    TEXT549 : BOOL ;	//TEXT N.549
    TEXT550 : BOOL ;	//TEXT N.550
    TEXT551 : BOOL ;	//TEXT N.551
    TEXT552 : BOOL ;	//TEXT N.552
    TEXT569 : BOOL ;	//TEXT N.569
    TEXT570 : BOOL ;	//TEXT N.570
    TEXT571 : BOOL ;	//TEXT N.571
    TEXT572 : BOOL ;	//TEXT N.572
    TEXT573 : BOOL ;	//TEXT N.573
    TEXT574 : BOOL ;	//TEXT N.574
    TEXT575 : BOOL ;	//TEXT N.575
    TEXT576 : BOOL ;	//TEXT N.576
    TEXT561 : BOOL ;	//TEXT N.561
    TEXT562 : BOOL ;	//TEXT N.562
    TEXT563 : BOOL ;	//TEXT N.563
    TEXT564 : BOOL ;	//TEXT N.564
    TEXT565 : BOOL ;	//TEXT N.565
    TEXT566 : BOOL ;	//TEXT N.566
    TEXT567 : BOOL ;	//TEXT N.567
    TEXT568 : BOOL ;	//TEXT N.568
    TEXT585 : BOOL ;	//TEXT N.585
    TEXT586 : BOOL ;	//TEXT N.586
    TEXT587 : BOOL ;	//TEXT N.587
    TEXT588 : BOOL ;	//TEXT N.588
    TEXT589 : BOOL ;	//TEXT N.589
    TEXT590 : BOOL ;	//TEXT N.590
    TEXT591 : BOOL ;	//TEXT N.591
    TEXT592 : BOOL ;	//TEXT N.592
    TEXT577 : BOOL ;	//TEXT N.577
    TEXT578 : BOOL ;	//TEXT N.578
    TEXT579 : BOOL ;	//TEXT N.579
    TEXT580 : BOOL ;	//TEXT N.580
    TEXT581 : BOOL ;	//TEXT N.581
    TEXT582 : BOOL ;	//TEXT N.582
    TEXT583 : BOOL ;	//TEXT N.583
    TEXT584 : BOOL ;	//TEXT N.584
    TEXT601 : BOOL ;	//TEXT N.601
    TEXT602 : BOOL ;	//TEXT N.602
    TEXT603 : BOOL ;	//TEXT N.603
    TEXT604 : BOOL ;	//TEXT N.604
    TEXT605 : BOOL ;	//TEXT N.605
    TEXT606 : BOOL ;	//TEXT N.606
    TEXT607 : BOOL ;	//TEXT N.607
    TEXT608 : BOOL ;	//TEXT N.608
    TEXT593 : BOOL ;	//TEXT N.593
    TEXT594 : BOOL ;	//TEXT N.594
    TEXT595 : BOOL ;	//TEXT N.595
    TEXT596 : BOOL ;	//TEXT N.596
    TEXT597 : BOOL ;	//TEXT N.597
    TEXT598 : BOOL ;	//TEXT N.598
    TEXT599 : BOOL ;	//TEXT N.599
    TEXT600 : BOOL ;	//TEXT N.600
    TEXT617 : BOOL ;	//TEXT N.617
    TEXT618 : BOOL ;	//TEXT N.618
    TEXT619 : BOOL ;	//TEXT N.619
    TEXT620 : BOOL ;	//TEXT N.620
    TEXT621 : BOOL ;	//TEXT N.621
    TEXT622 : BOOL ;	//TEXT N.622
    TEXT623 : BOOL ;	//TEXT N.623
    TEXT624 : BOOL ;	//TEXT N.624
    TEXT609 : BOOL ;	//TEXT N.609
    TEXT610 : BOOL ;	//TEXT N.610
    TEXT611 : BOOL ;	//TEXT N.611
    TEXT612 : BOOL ;	//TEXT N.612
    TEXT613 : BOOL ;	//TEXT N.613
    TEXT614 : BOOL ;	//TEXT N.614
    TEXT615 : BOOL ;	//TEXT N.615
    TEXT616 : BOOL ;	//TEXT N.616
    TEXT633 : BOOL ;	//TEXT N.633
    TEXT634 : BOOL ;	//TEXT N.634
    TEXT635 : BOOL ;	//TEXT N.635
    TEXT636 : BOOL ;	//TEXT N.636
    TEXT637 : BOOL ;	//TEXT N.637
    TEXT638 : BOOL ;	//TEXT N.638
    TEXT639 : BOOL ;	//TEXT N.639
    TEXT640 : BOOL ;	//TEXT N.640
    TEXT625 : BOOL ;	//TEXT N.625
    TEXT626 : BOOL ;	//TEXT N.626
    TEXT627 : BOOL ;	//TEXT N.627
    TEXT628 : BOOL ;	//TEXT N.628
    TEXT629 : BOOL ;	//TEXT N.629
    TEXT630 : BOOL ;	//TEXT N.630
    TEXT631 : BOOL ;	//TEXT N.631
    TEXT632 : BOOL ;	//TEXT N.632
   END_STRUCT ;
   PaginaDaVisualizzare : INT ;	//Number of page to display
   PaginaPrecedenteSetup : INT ;	//Number of page displayed before "Setup" page
   NumeroComandoManuale : INT ;	//Number of manual command
   BoschProgramManuale : BYTE ;	//Number of program of screwdriver in manual mode
   ServiceAsseSelezionato : BYTE ;	//Axis selected for movement in service mode (0=X; 1=Y; 2=Z; 3=C; 4=P)
   ServiceTipoJog : BYTE ;	//Kind of jog movement in service mode (0=continue; 1=incremental)
   ServiceFieldsDisplayed : BYTE ;	//Identify the fields to be displayed in service page
   TypePointTeachIn : BYTE ;	//Kind of screw in teach-in mode
   PointWeldingTeachIn : BYTE ;	//Identification of the screw in tech-in mode
   TeachInFieldsDisplayed : STRUCT 	//Identify the fields to be displayed in teach-in page
    Punto1Saldatura : BOOL ;
    Punto2Saldatura : BOOL ;
    Punto3Saldatura : BOOL ;
    Punto4Saldatura : BOOL ;
    Punto5Saldatura : BOOL ;
    Punto6Saldatura : BOOL ;
    Punto7Saldatura : BOOL ;
    Punto8Saldatura : BOOL ;
    Punto9Saldatura : BOOL ;
    Punto10Saldatura : BOOL ;
    Punto11Saldatura : BOOL ;
    Punto12Saldatura : BOOL ;
    Punto13Saldatura : BOOL ;
    PuntoVisione : BOOL ;
    Riserva1 : BOOL ;
    Riserva2 : BOOL ;
   END_STRUCT ;
   Target_Inc : DINT ;	//Target for the incremental movement
  END_STRUCT ;	
BEGIN
END_DATA_BLOCK

DATA_BLOCK "Timer"	// DB 20
VERSION : 0.1
  STRUCT
   TmrOutGas : S5TIME  := S5T#1M;
   TmrIgnition : S5TIME  := S5T#20S;
   TmrDelayWelding : S5TIME  := S5T#300MS;
   time1 : S5TIME ;
   time11 : S5TIME ;
   time12 : S5TIME ;
   time13 : S5TIME ;
   time14 : S5TIME ;
   time15 : S5TIME ;
   time16 : S5TIME ;
   time17 : S5TIME ;
   time18 : S5TIME ;
   time19 : S5TIME ;
   time110 : S5TIME ;
   time111 : S5TIME ;
   time112 : S5TIME ;
   time113 : S5TIME ;
   time114 : S5TIME ;
   time115 : S5TIME ;
   time116 : S5TIME ;
   Override : INT  := 20;
   riserva : INT ;
   riserva2 : INT ;
   Comp01_OK : BOOL ;
   Comp02_OK : BOOL ;
   Comp03_OK : BOOL ;
   Comp04_OK : BOOL ;
   Comp05_OK : BOOL ;
   Comp06_OK : BOOL ;
   Comp07_OK : BOOL ;
   Comp08_OK : BOOL ;
   Comp09_OK : BOOL ;
   Comp10_OK : BOOL ;
   Comp11_OK : BOOL ;
   Comp12_OK : BOOL ;
   Comp13_OK : BOOL ;
   Comp14_OK : BOOL ;
   Comp15_OK : BOOL ;
   Comp16_OK : BOOL ;
   OffsetX1 : DINT ;
   OffsetY1 : DINT ;
   okAletta1 : BOOL ;
   okAletta2 : BOOL ;
   okAletta3 : BOOL ;
   okAletta4 : BOOL ;
   okAletta5 : BOOL ;
   okAletta6 : BOOL ;
   okAletta7 : BOOL ;
   okAletta8 : BOOL ;
   okAletta9 : BOOL ;
   okAletta10 : BOOL ;
   okAletta11 : BOOL ;
   okAletta12 : BOOL ;
   okAletta13 : BOOL ;
   okAletta14 : BOOL ;
   okAletta15 : BOOL ;
   okAletta16 : BOOL ;
   okAletta17 : BOOL ;
   okAletta18 : BOOL ;
   okAletta19 : BOOL ;
   okAletta20 : BOOL ;
   CheckComponent : BOOL  := TRUE;	//Check component with tool 1 --> Disable ; 0 --> Enable
   CheckTelec : BOOL ;	//Check Component with Omron 1 --> Disable ; 0 --> Enable
   check1 : BOOL ;
   CheckTelecafter : BOOL ;	//Check Component with Omron 1 --> Disable ; 0 --> Enable
   okAletta1_PP : BOOL ;
   okAletta2_PP : BOOL ;
   okAletta3_PP : BOOL ;
   okAletta4_PP : BOOL ;
   okAletta5_PP : BOOL ;
   okAletta6_PP : BOOL ;
   okAletta7_PP : BOOL ;
   okAletta8_PP : BOOL ;
   okAletta9_PP : BOOL ;
   okAletta10_PP : BOOL ;
   okAletta11_PP : BOOL ;
   okAletta12_PP : BOOL ;
   okAletta13_PP : BOOL ;
   okAletta14_PP : BOOL ;
   okAletta15_PP : BOOL ;
   okAletta16_PP : BOOL ;
   okAletta17_PP : BOOL ;
   okAletta18_PP : BOOL ;
   okAletta19_PP : BOOL ;
   okAletta20_PP : BOOL ;
   NumberVane : INT ;
  END_STRUCT ;	
BEGIN
   TmrOutGas := S5T#1M;
   TmrIgnition := S5T#20S;
   TmrDelayWelding := S5T#300MS;
   Override := 100;
   OffsetX1 := L#350;
   OffsetY1 := L#400;
END_DATA_BLOCK

DATA_BLOCK "DBWork"	// DB 21
TITLE = Recipe of part in production
VERSION : 0.1
  STRUCT
   Famiglia : BYTE  := B#16#2;	//Type of family of product(2=Step2; 3=Step3)
   Turbo : BYTE  := B#16#1;	//Type of product
   Portapezzo1 : INT  := 1;	//Code of work rest 1
   Portapezzo2 : INT  := 1;	//Code of work rest 2
   TempoSaldatura : ARRAY  [1 .. 20 ] OF STRUCT
    Tempo : S5TIME  := S5T#1S;
   END_STRUCT ;
   CoordSaldatura : ARRAY  [1 .. 20 ] OF //Coordinates of points
   STRUCT
    X1 : DINT ;	//X coordinate of point
    Y1 : DINT ;	//Y coordinate of point
    X2 : DINT ;
    Y2 : DINT ;
   END_STRUCT ;
   EnableTelecamera : BOOL  := TRUE;
   PP : ARRAY  [1 .. 2 ] OF STRUCT
    Vuoto : BOOL ;
    Caricato : BOOL ;
    Bloccato : BOOL ;
    Fuori : BOOL ;
    Dentro : BOOL ;
    InLavorazione : BOOL ;
    Lavorato : BOOL ;
    Buono : BOOL ;
    Scarto : BOOL ;
    NumSaldaturaAtt : INT ;
   END_STRUCT ;
   NumeroAnomalie : DINT ;
   NumeroPezziProd : DINT ;
   NumeroSaldature : INT ;
   Riserva : DINT ;	//position X for camera check
   Riserva1 : DINT ;	//position Y for camera check
   RotationTable : BOOL ;	//angle rotation 1-->PP1 on welding; 0-->PP2 on Welding
   PointCamCheck : ARRAY  [1 .. 10 ] OF STRUCT
    x : DINT ;
    y : DINT ;
   END_STRUCT ;
  END_STRUCT ;	
BEGIN
   Famiglia := B#16#2;
   Turbo := B#16#1;
   Portapezzo1 := 1;
   Portapezzo2 := 1;
   TempoSaldatura[1].Tempo := S5T#1S;
   TempoSaldatura[2].Tempo := S5T#2S;
   TempoSaldatura[3].Tempo := S5T#1S;
   TempoSaldatura[4].Tempo := S5T#1S;
   TempoSaldatura[5].Tempo := S5T#1S;
   TempoSaldatura[6].Tempo := S5T#1S;
   TempoSaldatura[7].Tempo := S5T#1S;
   TempoSaldatura[8].Tempo := S5T#1S;
   TempoSaldatura[9].Tempo := S5T#1S;
   TempoSaldatura[10].Tempo := S5T#1S;
   TempoSaldatura[11].Tempo := S5T#1S;
   TempoSaldatura[12].Tempo := S5T#1S;
   TempoSaldatura[13].Tempo := S5T#1S;
   TempoSaldatura[14].Tempo := S5T#1S;
   TempoSaldatura[15].Tempo := S5T#1S;
   TempoSaldatura[16].Tempo := S5T#1S;
   TempoSaldatura[17].Tempo := S5T#1S;
   TempoSaldatura[18].Tempo := S5T#1S;
   TempoSaldatura[19].Tempo := S5T#1S;
   TempoSaldatura[20].Tempo := S5T#1S;
   CoordSaldatura[1].X1 := L#-60766;
   CoordSaldatura[1].Y1 := L#-86096;
   CoordSaldatura[1].X2 := L#-60406;
   CoordSaldatura[1].Y2 := L#-86246;
   CoordSaldatura[2].X1 := L#-46600;
   CoordSaldatura[2].Y1 := L#-81431;
   CoordSaldatura[2].X2 := L#-46422;
   CoordSaldatura[2].Y2 := L#-81523;
   CoordSaldatura[3].X1 := L#-29709;
   CoordSaldatura[3].Y1 := L#-81739;
   CoordSaldatura[3].X2 := L#-29405;
   CoordSaldatura[3].Y2 := L#-81809;
   CoordSaldatura[4].X1 := L#-16402;
   CoordSaldatura[4].Y1 := L#-86931;
   CoordSaldatura[4].X2 := L#-116220;
   CoordSaldatura[4].Y2 := L#-86961;
   CoordSaldatura[5].X1 := L#-11762;
   CoordSaldatura[5].Y1 := L#-95066;
   CoordSaldatura[5].X2 := L#-11500;
   CoordSaldatura[5].Y2 := L#-95199;
   CoordSaldatura[6].X1 := L#-17500;
   CoordSaldatura[6].Y1 := L#-102971;
   CoordSaldatura[6].X2 := L#-17415;
   CoordSaldatura[6].Y2 := L#-103088;
   CoordSaldatura[7].X1 := L#-31505;
   CoordSaldatura[7].Y1 := L#-107714;
   CoordSaldatura[7].X2 := L#-31400;
   CoordSaldatura[7].Y2 := L#-108200;
   CoordSaldatura[8].X1 := L#-48449;
   CoordSaldatura[8].Y1 := L#-107375;
   CoordSaldatura[8].X2 := L#-48367;
   CoordSaldatura[8].Y2 := L#-107501;
   CoordSaldatura[9].X1 := L#-61760;
   CoordSaldatura[9].Y1 := L#-102188;
   CoordSaldatura[9].X2 := L#-61561;
   CoordSaldatura[9].Y2 := L#-102300;
   CoordSaldatura[10].X1 := L#-66400;
   CoordSaldatura[10].Y1 := L#-94028;
   CoordSaldatura[10].Y2 := L#-94249;
   EnableTelecamera := TRUE;
END_DATA_BLOCK

DATA_BLOCK "coordinate"	// DB 22
VERSION : 0.1
  STRUCT
   CoordSaldaturaPP1 : ARRAY  [1 .. 20 ] OF //Coordinates of points
   STRUCT
    X1 : DINT ;	//X coordinate of point PP1
    Y1 : DINT ;	//Y coordinate of point PP1
    X2 : DINT ;
    Y2 : DINT ;
   END_STRUCT ;
   CoordSaldaturaPP2 : ARRAY  [1 .. 20 ] OF //Coordinates of points
   STRUCT
    X1 : DINT ;	//X coordinate of point PP2
    Y1 : DINT ;	//Y coordinate of point PP2
    X2 : DINT ;
    Y2 : DINT ;
   END_STRUCT ;
   CoordSaldaturaPP3 : ARRAY  [1 .. 20 ] OF //Coordinates of points
   STRUCT
    X1 : DINT ;	//X coordinate of point PP3
    Y1 : DINT ;	//Y coordinate of point PP3
    X2 : DINT ;
    Y2 : DINT ;
   END_STRUCT ;
   CoordSaldaturaPP4 : ARRAY  [1 .. 20 ] OF //Coordinates of points
   STRUCT
    X1 : DINT ;	//X coordinate of point PP4
    Y1 : DINT ;	//Y coordinate of point PP4
    X2 : DINT ;
    Y2 : DINT ;
   END_STRUCT ;
   CoordSaldaturaPP5 : ARRAY  [1 .. 20 ] OF //Coordinates of points
   STRUCT
    X1 : DINT ;	//X coordinate of point PP5
    Y1 : DINT ;	//Y coordinate of point PP5
    X2 : DINT ;
    Y2 : DINT ;
   END_STRUCT ;
   CoordSaldaturaPP6 : ARRAY  [1 .. 20 ] OF STRUCT
    X1 : DINT ;
    Y1 : DINT ;
    X2 : DINT ;
    Y2 : DINT ;
   END_STRUCT ;
   CoordSaldaturaPP7 : ARRAY  [1 .. 20 ] OF STRUCT
    X1 : DINT ;
    Y1 : DINT ;
    X2 : DINT ;
    Y2 : DINT ;
   END_STRUCT ;
   CoordSaldaturaPP8 : ARRAY  [1 .. 20 ] OF STRUCT
    X1 : DINT ;
    Y1 : DINT ;
    X2 : DINT ;
    Y2 : DINT ;
   END_STRUCT ;
   CoordSaldaturaPP9 : ARRAY  [1 .. 20 ] OF STRUCT
    X1 : DINT ;
    Y1 : DINT ;
    X2 : DINT ;
    Y2 : DINT ;
   END_STRUCT ;
   CoordSaldaturaPP10 : ARRAY  [1 .. 20 ] OF STRUCT
    X1 : DINT ;
    Y1 : DINT ;
    X2 : DINT ;
    Y2 : DINT ;
   END_STRUCT ;
   CoordSaldaturaPP11 : ARRAY  [1 .. 20 ] OF STRUCT
    X1 : DINT ;
    Y1 : DINT ;
    X2 : DINT ;
    Y2 : DINT ;
   END_STRUCT ;
   CoordSaldaturaPP12 : ARRAY  [1 .. 20 ] OF STRUCT
    X1 : DINT ;
    Y1 : DINT ;
    X2 : DINT ;
    Y2 : DINT ;
   END_STRUCT ;
   CoordSaldaturaPP13 : ARRAY  [1 .. 20 ] OF STRUCT
    X1 : DINT ;
    Y1 : DINT ;
    X2 : DINT ;
    Y2 : DINT ;
   END_STRUCT ;
   CoordSaldaturaPP14 : ARRAY  [1 .. 20 ] OF STRUCT
    X1 : DINT ;
    Y1 : DINT ;
    X2 : DINT ;
    Y2 : DINT ;
   END_STRUCT ;
   CoordSaldaturaPP15 : ARRAY  [1 .. 20 ] OF STRUCT
    X1 : DINT ;
    Y1 : DINT ;
    X2 : DINT ;
    Y2 : DINT ;
   END_STRUCT ;
   CoordSaldaturaPP16 : ARRAY  [1 .. 20 ] OF STRUCT
    X1 : DINT ;
    Y1 : DINT ;
    X2 : DINT ;
    Y2 : DINT ;
   END_STRUCT ;
   CoordSaldaturaPP17 : ARRAY  [1 .. 20 ] OF STRUCT
    X1 : DINT ;
    Y1 : DINT ;
    X2 : DINT ;
    Y2 : DINT ;
   END_STRUCT ;
   CoordSaldaturaPP18 : ARRAY  [1 .. 20 ] OF STRUCT
    X1 : DINT ;
    Y1 : DINT ;
    X2 : DINT ;
    Y2 : DINT ;
   END_STRUCT ;
   CoordSaldaturaPP19 : ARRAY  [1 .. 20 ] OF STRUCT
    X1 : DINT ;
    Y1 : DINT ;
    X2 : DINT ;
    Y2 : DINT ;
   END_STRUCT ;
   CoordSaldaturaPP20 : ARRAY  [1 .. 20 ] OF STRUCT
    X1 : DINT ;
    Y1 : DINT ;
    X2 : DINT ;
    Y2 : DINT ;
   END_STRUCT ;
   CoordinateCam_PP1 : ARRAY  [1 .. 10 ] OF STRUCT
    X : DINT ;	//X coordinate of point cam PP1
    Y : DINT ;	//X coordinate of point cam PP1
   END_STRUCT ;
   CoordinateCam_PP2 : ARRAY  [1 .. 10 ] OF STRUCT
    X : DINT ;	//X coordinate of point cam PP1
    Y : DINT ;	//X coordinate of point cam PP1
   END_STRUCT ;
   CoordinateCam_PP3 : ARRAY  [1 .. 10 ] OF STRUCT
    X : DINT ;	//X coordinate of point cam PP1
    Y : DINT ;	//X coordinate of point cam PP1
   END_STRUCT ;
   CoordinateCam_PP4 : ARRAY  [1 .. 10 ] OF STRUCT
    X : DINT ;	//X coordinate of point cam PP1
    Y : DINT ;	//X coordinate of point cam PP1
   END_STRUCT ;
   CoordinateCam_PP5 : ARRAY  [1 .. 10 ] OF STRUCT
    X : DINT ;	//X coordinate of point cam PP1
    Y : DINT ;	//X coordinate of point cam PP1
   END_STRUCT ;
   CoordinateCam_PP6 : ARRAY  [1 .. 10 ] OF STRUCT
    X : DINT ;	//X coordinate of point cam PP1
    Y : DINT ;	//X coordinate of point cam PP1
   END_STRUCT ;
   CoordinateCam_PP7 : ARRAY  [1 .. 10 ] OF STRUCT
    X : DINT ;	//X coordinate of point cam PP1
    Y : DINT ;	//X coordinate of point cam PP1
   END_STRUCT ;
   CoordinateCam_PP8 : ARRAY  [1 .. 10 ] OF STRUCT
    X : DINT ;	//X coordinate of point cam PP1
    Y : DINT ;	//X coordinate of point cam PP1
   END_STRUCT ;
   CoordinateCam_PP9 : ARRAY  [1 .. 10 ] OF STRUCT
    X : DINT ;	//X coordinate of point cam PP1
    Y : DINT ;	//X coordinate of point cam PP1
   END_STRUCT ;
   CoordinateCam_PP10 : ARRAY  [1 .. 10 ] OF STRUCT
    X : DINT ;	//X coordinate of point cam PP1
    Y : DINT ;	//X coordinate of point cam PP1
   END_STRUCT ;
   CoordinateCam_PP11 : ARRAY  [1 .. 10 ] OF STRUCT
    X : DINT ;	//X coordinate of point cam PP1
    Y : DINT ;	//X coordinate of point cam PP1
   END_STRUCT ;
   CoordinateCam_PP12 : ARRAY  [1 .. 10 ] OF STRUCT
    X : DINT ;	//X coordinate of point cam PP1
    Y : DINT ;	//X coordinate of point cam PP1
   END_STRUCT ;
   CoordinateCam_PP13 : ARRAY  [1 .. 10 ] OF STRUCT
    X : DINT ;	//X coordinate of point cam PP1
    Y : DINT ;	//X coordinate of point cam PP1
   END_STRUCT ;
   CoordinateCam_PP14 : ARRAY  [1 .. 10 ] OF STRUCT
    X : DINT ;	//X coordinate of point cam PP1
    Y : DINT ;	//X coordinate of point cam PP1
   END_STRUCT ;
   CoordinateCam_PP15 : ARRAY  [1 .. 10 ] OF STRUCT
    X : DINT ;	//X coordinate of point cam PP1
    Y : DINT ;	//X coordinate of point cam PP1
   END_STRUCT ;
   CoordinateCam_PP16 : ARRAY  [1 .. 10 ] OF STRUCT
    X : DINT ;	//X coordinate of point cam PP1
    Y : DINT ;	//X coordinate of point cam PP1
   END_STRUCT ;
   CoordinateCam_PP17 : ARRAY  [1 .. 10 ] OF STRUCT
    X : DINT ;	//X coordinate of point cam PP1
    Y : DINT ;	//X coordinate of point cam PP1
   END_STRUCT ;
   CoordinateCam_PP18 : ARRAY  [1 .. 10 ] OF STRUCT
    X : DINT ;	//X coordinate of point cam PP1
    Y : DINT ;	//X coordinate of point cam PP1
   END_STRUCT ;
   CoordinateCam_PP19 : ARRAY  [1 .. 10 ] OF STRUCT
    X : DINT ;	//X coordinate of point cam PP1
    Y : DINT ;	//X coordinate of point cam PP1
   END_STRUCT ;
   CoordinateCam_PP20 : ARRAY  [1 .. 10 ] OF STRUCT
    X : DINT ;	//X coordinate of point cam PP1
    Y : DINT ;	//X coordinate of point cam PP1
   END_STRUCT ;
   NumeroSaldaturePP1 : INT ;
   NumeroSaldaturePP2 : INT ;
   NumeroSaldaturePP3 : INT ;
   NumeroSaldaturePP4 : INT ;
   NumeroSaldaturePP5 : INT ;
   NumeroSaldaturePP6 : INT ;
   NumeroSaldaturePP7 : INT ;
   NumeroSaldaturePP8 : INT ;
   NumeroSaldaturePP9 : INT ;
   NumeroSaldaturePP10 : INT ;
   NumeroSaldaturePP11 : INT ;
   NumeroSaldaturePP12 : INT ;
   NumeroSaldaturePP13 : INT ;
   NumeroSaldaturePP14 : INT ;
   NumeroSaldaturePP15 : INT ;
   NumeroSaldaturePP16 : INT ;
   NumeroSaldaturePP17 : INT ;
   NumeroSaldaturePP18 : INT ;
   NumeroSaldaturePP19 : INT ;
   NumeroSaldaturePP20 : INT ;
   TimeWeldingPP1 : ARRAY  [1 .. 20 ] OF STRUCT
    Tempo : S5TIME  := S5T#1S;
   END_STRUCT ;
   TimeWeldingPP2 : ARRAY  [1 .. 20 ] OF STRUCT
    Tempo : S5TIME  := S5T#1S;
   END_STRUCT ;
   TimeWeldingPP3 : ARRAY  [1 .. 20 ] OF STRUCT
    Tempo : S5TIME  := S5T#1S;
   END_STRUCT ;
   TimeWeldingPP4 : ARRAY  [1 .. 20 ] OF STRUCT
    Tempo : S5TIME  := S5T#1S;
   END_STRUCT ;
   TimeWeldingPP5 : ARRAY  [1 .. 20 ] OF STRUCT
    Tempo : S5TIME  := S5T#1S;
   END_STRUCT ;
   TimeWeldingPP6 : ARRAY  [1 .. 20 ] OF STRUCT
    Tempo : S5TIME  := S5T#1S;
   END_STRUCT ;
   TimeWeldingPP7 : ARRAY  [1 .. 20 ] OF STRUCT
    Tempo : S5TIME  := S5T#1S;
   END_STRUCT ;
   TimeWeldingPP8 : ARRAY  [1 .. 20 ] OF STRUCT
    Tempo : S5TIME  := S5T#1S;
   END_STRUCT ;
   TimeWeldingPP9 : ARRAY  [1 .. 20 ] OF STRUCT
    Tempo : S5TIME  := S5T#1S;
   END_STRUCT ;
   TimeWeldingPP10 : ARRAY  [1 .. 20 ] OF STRUCT
    Tempo : S5TIME  := S5T#1S;
   END_STRUCT ;
   TimeWeldingPP11 : ARRAY  [1 .. 20 ] OF STRUCT
    Tempo : S5TIME  := S5T#1S;
   END_STRUCT ;
   TimeWeldingPP12 : ARRAY  [1 .. 20 ] OF STRUCT
    Tempo : S5TIME  := S5T#1S;
   END_STRUCT ;
   TimeWeldingPP13 : ARRAY  [1 .. 20 ] OF STRUCT
    Tempo : S5TIME  := S5T#1S;
   END_STRUCT ;
   TimeWeldingPP14 : ARRAY  [1 .. 20 ] OF STRUCT
    Tempo : S5TIME  := S5T#1S;
   END_STRUCT ;
   TimeWeldingPP15 : ARRAY  [1 .. 20 ] OF STRUCT
    Tempo : S5TIME  := S5T#1S;
   END_STRUCT ;
   TimeWeldingPP16 : ARRAY  [1 .. 20 ] OF STRUCT
    Tempo : S5TIME  := S5T#1S;
   END_STRUCT ;
   TimeWeldingPP17 : ARRAY  [1 .. 20 ] OF STRUCT
    Tempo : S5TIME  := S5T#1S;
   END_STRUCT ;
   TimeWeldingPP18 : ARRAY  [1 .. 20 ] OF STRUCT
    Tempo : S5TIME  := S5T#1S;
   END_STRUCT ;
   TimeWeldingPP19 : ARRAY  [1 .. 20 ] OF STRUCT
    Tempo : S5TIME  := S5T#1S;
   END_STRUCT ;
   TimeWeldingPP20 : ARRAY  [1 .. 20 ] OF STRUCT
    Tempo : S5TIME  := S5T#1S;
   END_STRUCT ;
  END_STRUCT ;	
BEGIN
   CoordSaldaturaPP1[1].X1 := L#-60530;
   CoordSaldaturaPP1[1].Y1 := L#-172340;
   CoordSaldaturaPP1[1].X2 := L#-60530;
   CoordSaldaturaPP1[1].Y2 := L#-172340;
   CoordSaldaturaPP1[2].X1 := L#-46530;
   CoordSaldaturaPP1[2].Y1 := L#-162870;
   CoordSaldaturaPP1[2].X2 := L#-46530;
   CoordSaldaturaPP1[2].Y2 := L#-162870;
   CoordSaldaturaPP1[3].X1 := L#-29630;
   CoordSaldaturaPP1[3].Y1 := L#-163440;
   CoordSaldaturaPP1[3].X2 := L#-29630;
   CoordSaldaturaPP1[3].Y2 := L#-163440;
   CoordSaldaturaPP1[4].X1 := L#-16300;
   CoordSaldaturaPP1[4].Y1 := L#-173820;
   CoordSaldaturaPP1[4].X2 := L#-16300;
   CoordSaldaturaPP1[4].Y2 := L#-173820;
   CoordSaldaturaPP1[5].X1 := L#-11620;
   CoordSaldaturaPP1[5].Y1 := L#-190070;
   CoordSaldaturaPP1[5].X2 := L#-11620;
   CoordSaldaturaPP1[5].Y2 := L#-190070;
   CoordSaldaturaPP1[6].X1 := L#-17370;
   CoordSaldaturaPP1[6].Y1 := L#-205960;
   CoordSaldaturaPP1[6].X2 := L#-17370;
   CoordSaldaturaPP1[6].Y2 := L#-205960;
   CoordSaldaturaPP1[7].X1 := L#-31370;
   CoordSaldaturaPP1[7].Y1 := L#-215430;
   CoordSaldaturaPP1[7].X2 := L#-31370;
   CoordSaldaturaPP1[7].Y2 := L#-215430;
   CoordSaldaturaPP1[8].X1 := L#-48270;
   CoordSaldaturaPP1[8].Y1 := L#-214860;
   CoordSaldaturaPP1[8].X2 := L#-48270;
   CoordSaldaturaPP1[8].Y2 := L#-214860;
   CoordSaldaturaPP1[9].X1 := L#-61600;
   CoordSaldaturaPP1[9].Y1 := L#-204480;
   CoordSaldaturaPP1[9].X2 := L#-61600;
   CoordSaldaturaPP1[9].Y2 := L#-204480;
   CoordSaldaturaPP1[10].X1 := L#-66280;
   CoordSaldaturaPP1[10].Y1 := L#-188230;
   CoordSaldaturaPP1[10].X2 := L#-66280;
   CoordSaldaturaPP1[10].Y2 := L#-188230;
   CoordSaldaturaPP6[1].X1 := L#-24431;
   CoordSaldaturaPP6[1].Y1 := L#-211667;
   CoordSaldaturaPP6[1].X2 := L#-24468;
   CoordSaldaturaPP6[1].Y2 := L#-211634;
   CoordSaldaturaPP6[2].X1 := L#-13011;
   CoordSaldaturaPP6[2].Y1 := L#-199436;
   CoordSaldaturaPP6[2].X2 := L#-12856;
   CoordSaldaturaPP6[2].Y2 := L#-199488;
   CoordSaldaturaPP6[3].X1 := L#-9745;
   CoordSaldaturaPP6[3].Y1 := L#-183598;
   CoordSaldaturaPP6[3].X2 := L#-9756;
   CoordSaldaturaPP6[3].Y2 := L#-183663;
   CoordSaldaturaPP6[4].X1 := L#-16203;
   CoordSaldaturaPP6[4].Y1 := L#-168150;
   CoordSaldaturaPP6[4].X2 := L#-16141;
   CoordSaldaturaPP6[4].Y2 := L#-168156;
   CoordSaldaturaPP6[5].X1 := L#-29434;
   CoordSaldaturaPP6[5].Y1 := L#-158429;
   CoordSaldaturaPP6[5].X2 := L#-29472;
   CoordSaldaturaPP6[5].Y2 := L#-158489;
   CoordSaldaturaPP6[6].X1 := L#-46262;
   CoordSaldaturaPP6[6].Y1 := L#-157658;
   CoordSaldaturaPP6[6].X2 := L#-46155;
   CoordSaldaturaPP6[6].Y2 := L#-157716;
   CoordSaldaturaPP6[7].X1 := L#-60740;
   CoordSaldaturaPP6[7].Y1 := L#-166127;
   CoordSaldaturaPP6[7].X2 := L#-60564;
   CoordSaldaturaPP6[7].Y2 := L#-166296;
   CoordSaldaturaPP6[8].X1 := L#-68335;
   CoordSaldaturaPP6[8].Y1 := L#-180765;
   CoordSaldaturaPP6[8].X2 := L#-68026;
   CoordSaldaturaPP6[8].Y2 := L#-180787;
   CoordSaldaturaPP6[9].X1 := L#-66468;
   CoordSaldaturaPP6[9].Y1 := L#-197254;
   CoordSaldaturaPP6[9].X2 := L#-66217;
   CoordSaldaturaPP6[9].Y2 := L#-197398;
   CoordSaldaturaPP6[10].X1 := L#-56162;
   CoordSaldaturaPP6[10].Y1 := L#-210332;
   CoordSaldaturaPP6[10].X2 := L#-56200;
   CoordSaldaturaPP6[10].Y2 := L#-210331;
   CoordSaldaturaPP6[11].X1 := L#-40981;
   CoordSaldaturaPP6[11].Y1 := L#-215911;
   CoordSaldaturaPP6[11].X2 := L#-40587;
   CoordSaldaturaPP6[11].Y2 := L#-215681;
   CoordSaldaturaPP11[1].X1 := L#-24431;
   CoordSaldaturaPP11[1].Y1 := L#-211667;
   CoordSaldaturaPP11[1].X2 := L#-24468;
   CoordSaldaturaPP11[1].Y2 := L#-211634;
   CoordSaldaturaPP11[2].X1 := L#-13011;
   CoordSaldaturaPP11[2].Y1 := L#-199436;
   CoordSaldaturaPP11[2].X2 := L#-12856;
   CoordSaldaturaPP11[2].Y2 := L#-199488;
   CoordSaldaturaPP11[3].X1 := L#-9745;
   CoordSaldaturaPP11[3].Y1 := L#-183598;
   CoordSaldaturaPP11[3].X2 := L#-9786;
   CoordSaldaturaPP11[3].Y2 := L#-183663;
   CoordSaldaturaPP11[4].X1 := L#-16203;
   CoordSaldaturaPP11[4].Y1 := L#-168150;
   CoordSaldaturaPP11[4].X2 := L#-16141;
   CoordSaldaturaPP11[4].Y2 := L#-168156;
   CoordSaldaturaPP11[5].X1 := L#-29434;
   CoordSaldaturaPP11[5].Y1 := L#-158429;
   CoordSaldaturaPP11[5].X2 := L#-29472;
   CoordSaldaturaPP11[5].Y2 := L#-158489;
   CoordSaldaturaPP11[6].X1 := L#-46262;
   CoordSaldaturaPP11[6].Y1 := L#-157658;
   CoordSaldaturaPP11[6].X2 := L#-46155;
   CoordSaldaturaPP11[6].Y2 := L#-157716;
   CoordSaldaturaPP11[7].X1 := L#-60740;
   CoordSaldaturaPP11[7].Y1 := L#-166127;
   CoordSaldaturaPP11[7].X2 := L#-60564;
   CoordSaldaturaPP11[7].Y2 := L#-166296;
   CoordSaldaturaPP11[8].X1 := L#-68335;
   CoordSaldaturaPP11[8].Y1 := L#-180765;
   CoordSaldaturaPP11[8].X2 := L#-68026;
   CoordSaldaturaPP11[8].Y2 := L#-180787;
   CoordSaldaturaPP11[9].X1 := L#-66468;
   CoordSaldaturaPP11[9].Y1 := L#-197254;
   CoordSaldaturaPP11[9].X2 := L#-66217;
   CoordSaldaturaPP11[9].Y2 := L#-197398;
   CoordSaldaturaPP11[10].X1 := L#-56162;
   CoordSaldaturaPP11[10].Y1 := L#-210332;
   CoordSaldaturaPP11[10].X2 := L#-56200;
   CoordSaldaturaPP11[10].Y2 := L#-210331;
   CoordSaldaturaPP11[11].X1 := L#-40981;
   CoordSaldaturaPP11[11].Y1 := L#-215911;
   CoordSaldaturaPP11[11].X2 := L#-40587;
   CoordSaldaturaPP11[11].Y2 := L#-215681;
   CoordinateCam_PP1[1].X := L#7915;
   CoordinateCam_PP1[1].Y := L#-68282;
   NumeroSaldaturePP1 := 10;
   TimeWeldingPP1[1].Tempo := S5T#1S;
   TimeWeldingPP1[2].Tempo := S5T#2S;
   TimeWeldingPP1[3].Tempo := S5T#1S;
   TimeWeldingPP1[4].Tempo := S5T#1S;
   TimeWeldingPP1[5].Tempo := S5T#1S;
   TimeWeldingPP1[6].Tempo := S5T#1S;
   TimeWeldingPP1[7].Tempo := S5T#1S;
   TimeWeldingPP1[8].Tempo := S5T#1S;
   TimeWeldingPP1[9].Tempo := S5T#1S;
   TimeWeldingPP1[10].Tempo := S5T#1S;
   TimeWeldingPP1[11].Tempo := S5T#1S;
   TimeWeldingPP1[12].Tempo := S5T#1S;
   TimeWeldingPP1[13].Tempo := S5T#1S;
   TimeWeldingPP1[14].Tempo := S5T#1S;
   TimeWeldingPP1[15].Tempo := S5T#1S;
   TimeWeldingPP1[16].Tempo := S5T#1S;
   TimeWeldingPP1[17].Tempo := S5T#1S;
   TimeWeldingPP1[18].Tempo := S5T#1S;
   TimeWeldingPP1[19].Tempo := S5T#1S;
   TimeWeldingPP1[20].Tempo := S5T#1S;
   TimeWeldingPP2[1].Tempo := S5T#1S;
   TimeWeldingPP2[2].Tempo := S5T#1S;
   TimeWeldingPP2[3].Tempo := S5T#1S;
   TimeWeldingPP2[4].Tempo := S5T#1S;
   TimeWeldingPP2[5].Tempo := S5T#1S;
   TimeWeldingPP2[6].Tempo := S5T#1S;
   TimeWeldingPP2[7].Tempo := S5T#1S;
   TimeWeldingPP2[8].Tempo := S5T#1S;
   TimeWeldingPP2[9].Tempo := S5T#1S;
   TimeWeldingPP2[10].Tempo := S5T#1S;
   TimeWeldingPP2[11].Tempo := S5T#1S;
   TimeWeldingPP2[12].Tempo := S5T#1S;
   TimeWeldingPP2[13].Tempo := S5T#1S;
   TimeWeldingPP2[14].Tempo := S5T#1S;
   TimeWeldingPP2[15].Tempo := S5T#1S;
   TimeWeldingPP2[16].Tempo := S5T#1S;
   TimeWeldingPP2[17].Tempo := S5T#1S;
   TimeWeldingPP2[18].Tempo := S5T#1S;
   TimeWeldingPP2[19].Tempo := S5T#1S;
   TimeWeldingPP2[20].Tempo := S5T#1S;
   TimeWeldingPP3[1].Tempo := S5T#1S;
   TimeWeldingPP3[2].Tempo := S5T#1S;
   TimeWeldingPP3[3].Tempo := S5T#1S;
   TimeWeldingPP3[4].Tempo := S5T#1S;
   TimeWeldingPP3[5].Tempo := S5T#1S;
   TimeWeldingPP3[6].Tempo := S5T#1S;
   TimeWeldingPP3[7].Tempo := S5T#1S;
   TimeWeldingPP3[8].Tempo := S5T#1S;
   TimeWeldingPP3[9].Tempo := S5T#1S;
   TimeWeldingPP3[10].Tempo := S5T#1S;
   TimeWeldingPP3[11].Tempo := S5T#1S;
   TimeWeldingPP3[12].Tempo := S5T#1S;
   TimeWeldingPP3[13].Tempo := S5T#1S;
   TimeWeldingPP3[14].Tempo := S5T#1S;
   TimeWeldingPP3[15].Tempo := S5T#1S;
   TimeWeldingPP3[16].Tempo := S5T#1S;
   TimeWeldingPP3[17].Tempo := S5T#1S;
   TimeWeldingPP3[18].Tempo := S5T#1S;
   TimeWeldingPP3[19].Tempo := S5T#1S;
   TimeWeldingPP3[20].Tempo := S5T#1S;
   TimeWeldingPP4[1].Tempo := S5T#1S;
   TimeWeldingPP4[2].Tempo := S5T#1S;
   TimeWeldingPP4[3].Tempo := S5T#1S;
   TimeWeldingPP4[4].Tempo := S5T#1S;
   TimeWeldingPP4[5].Tempo := S5T#1S;
   TimeWeldingPP4[6].Tempo := S5T#1S;
   TimeWeldingPP4[7].Tempo := S5T#1S;
   TimeWeldingPP4[8].Tempo := S5T#1S;
   TimeWeldingPP4[9].Tempo := S5T#1S;
   TimeWeldingPP4[10].Tempo := S5T#1S;
   TimeWeldingPP4[11].Tempo := S5T#1S;
   TimeWeldingPP4[12].Tempo := S5T#1S;
   TimeWeldingPP4[13].Tempo := S5T#1S;
   TimeWeldingPP4[14].Tempo := S5T#1S;
   TimeWeldingPP4[15].Tempo := S5T#1S;
   TimeWeldingPP4[16].Tempo := S5T#1S;
   TimeWeldingPP4[17].Tempo := S5T#1S;
   TimeWeldingPP4[18].Tempo := S5T#1S;
   TimeWeldingPP4[19].Tempo := S5T#1S;
   TimeWeldingPP4[20].Tempo := S5T#1S;
   TimeWeldingPP5[1].Tempo := S5T#1S;
   TimeWeldingPP5[2].Tempo := S5T#1S;
   TimeWeldingPP5[3].Tempo := S5T#1S;
   TimeWeldingPP5[4].Tempo := S5T#1S;
   TimeWeldingPP5[5].Tempo := S5T#1S;
   TimeWeldingPP5[6].Tempo := S5T#1S;
   TimeWeldingPP5[7].Tempo := S5T#1S;
   TimeWeldingPP5[8].Tempo := S5T#1S;
   TimeWeldingPP5[9].Tempo := S5T#1S;
   TimeWeldingPP5[10].Tempo := S5T#1S;
   TimeWeldingPP5[11].Tempo := S5T#1S;
   TimeWeldingPP5[12].Tempo := S5T#1S;
   TimeWeldingPP5[13].Tempo := S5T#1S;
   TimeWeldingPP5[14].Tempo := S5T#1S;
   TimeWeldingPP5[15].Tempo := S5T#1S;
   TimeWeldingPP5[16].Tempo := S5T#1S;
   TimeWeldingPP5[17].Tempo := S5T#1S;
   TimeWeldingPP5[18].Tempo := S5T#1S;
   TimeWeldingPP5[19].Tempo := S5T#1S;
   TimeWeldingPP5[20].Tempo := S5T#1S;
   TimeWeldingPP6[1].Tempo := S5T#1S;
   TimeWeldingPP6[2].Tempo := S5T#1S;
   TimeWeldingPP6[3].Tempo := S5T#1S;
   TimeWeldingPP6[4].Tempo := S5T#1S;
   TimeWeldingPP6[5].Tempo := S5T#1S;
   TimeWeldingPP6[6].Tempo := S5T#1S;
   TimeWeldingPP6[7].Tempo := S5T#1S;
   TimeWeldingPP6[8].Tempo := S5T#1S;
   TimeWeldingPP6[9].Tempo := S5T#1S;
   TimeWeldingPP6[10].Tempo := S5T#1S;
   TimeWeldingPP6[11].Tempo := S5T#1S;
   TimeWeldingPP6[12].Tempo := S5T#1S;
   TimeWeldingPP6[13].Tempo := S5T#1S;
   TimeWeldingPP6[14].Tempo := S5T#1S;
   TimeWeldingPP6[15].Tempo := S5T#1S;
   TimeWeldingPP6[16].Tempo := S5T#1S;
   TimeWeldingPP6[17].Tempo := S5T#1S;
   TimeWeldingPP6[18].Tempo := S5T#1S;
   TimeWeldingPP6[19].Tempo := S5T#1S;
   TimeWeldingPP6[20].Tempo := S5T#1S;
   TimeWeldingPP7[1].Tempo := S5T#1S;
   TimeWeldingPP7[2].Tempo := S5T#1S;
   TimeWeldingPP7[3].Tempo := S5T#1S;
   TimeWeldingPP7[4].Tempo := S5T#1S;
   TimeWeldingPP7[5].Tempo := S5T#1S;
   TimeWeldingPP7[6].Tempo := S5T#1S;
   TimeWeldingPP7[7].Tempo := S5T#1S;
   TimeWeldingPP7[8].Tempo := S5T#1S;
   TimeWeldingPP7[9].Tempo := S5T#1S;
   TimeWeldingPP7[10].Tempo := S5T#1S;
   TimeWeldingPP7[11].Tempo := S5T#1S;
   TimeWeldingPP7[12].Tempo := S5T#1S;
   TimeWeldingPP7[13].Tempo := S5T#1S;
   TimeWeldingPP7[14].Tempo := S5T#1S;
   TimeWeldingPP7[15].Tempo := S5T#1S;
   TimeWeldingPP7[16].Tempo := S5T#1S;
   TimeWeldingPP7[17].Tempo := S5T#1S;
   TimeWeldingPP7[18].Tempo := S5T#1S;
   TimeWeldingPP7[19].Tempo := S5T#1S;
   TimeWeldingPP7[20].Tempo := S5T#1S;
   TimeWeldingPP8[1].Tempo := S5T#1S;
   TimeWeldingPP8[2].Tempo := S5T#1S;
   TimeWeldingPP8[3].Tempo := S5T#1S;
   TimeWeldingPP8[4].Tempo := S5T#1S;
   TimeWeldingPP8[5].Tempo := S5T#1S;
   TimeWeldingPP8[6].Tempo := S5T#1S;
   TimeWeldingPP8[7].Tempo := S5T#1S;
   TimeWeldingPP8[8].Tempo := S5T#1S;
   TimeWeldingPP8[9].Tempo := S5T#1S;
   TimeWeldingPP8[10].Tempo := S5T#1S;
   TimeWeldingPP8[11].Tempo := S5T#1S;
   TimeWeldingPP8[12].Tempo := S5T#1S;
   TimeWeldingPP8[13].Tempo := S5T#1S;
   TimeWeldingPP8[14].Tempo := S5T#1S;
   TimeWeldingPP8[15].Tempo := S5T#1S;
   TimeWeldingPP8[16].Tempo := S5T#1S;
   TimeWeldingPP8[17].Tempo := S5T#1S;
   TimeWeldingPP8[18].Tempo := S5T#1S;
   TimeWeldingPP8[19].Tempo := S5T#1S;
   TimeWeldingPP8[20].Tempo := S5T#1S;
   TimeWeldingPP9[1].Tempo := S5T#1S;
   TimeWeldingPP9[2].Tempo := S5T#1S;
   TimeWeldingPP9[3].Tempo := S5T#1S;
   TimeWeldingPP9[4].Tempo := S5T#1S;
   TimeWeldingPP9[5].Tempo := S5T#1S;
   TimeWeldingPP9[6].Tempo := S5T#1S;
   TimeWeldingPP9[7].Tempo := S5T#1S;
   TimeWeldingPP9[8].Tempo := S5T#1S;
   TimeWeldingPP9[9].Tempo := S5T#1S;
   TimeWeldingPP9[10].Tempo := S5T#1S;
   TimeWeldingPP9[11].Tempo := S5T#1S;
   TimeWeldingPP9[12].Tempo := S5T#1S;
   TimeWeldingPP9[13].Tempo := S5T#1S;
   TimeWeldingPP9[14].Tempo := S5T#1S;
   TimeWeldingPP9[15].Tempo := S5T#1S;
   TimeWeldingPP9[16].Tempo := S5T#1S;
   TimeWeldingPP9[17].Tempo := S5T#1S;
   TimeWeldingPP9[18].Tempo := S5T#1S;
   TimeWeldingPP9[19].Tempo := S5T#1S;
   TimeWeldingPP9[20].Tempo := S5T#1S;
   TimeWeldingPP10[1].Tempo := S5T#1S;
   TimeWeldingPP10[2].Tempo := S5T#1S;
   TimeWeldingPP10[3].Tempo := S5T#1S;
   TimeWeldingPP10[4].Tempo := S5T#1S;
   TimeWeldingPP10[5].Tempo := S5T#1S;
   TimeWeldingPP10[6].Tempo := S5T#1S;
   TimeWeldingPP10[7].Tempo := S5T#1S;
   TimeWeldingPP10[8].Tempo := S5T#1S;
   TimeWeldingPP10[9].Tempo := S5T#1S;
   TimeWeldingPP10[10].Tempo := S5T#1S;
   TimeWeldingPP10[11].Tempo := S5T#1S;
   TimeWeldingPP10[12].Tempo := S5T#1S;
   TimeWeldingPP10[13].Tempo := S5T#1S;
   TimeWeldingPP10[14].Tempo := S5T#1S;
   TimeWeldingPP10[15].Tempo := S5T#1S;
   TimeWeldingPP10[16].Tempo := S5T#1S;
   TimeWeldingPP10[17].Tempo := S5T#1S;
   TimeWeldingPP10[18].Tempo := S5T#1S;
   TimeWeldingPP10[19].Tempo := S5T#1S;
   TimeWeldingPP10[20].Tempo := S5T#1S;
   TimeWeldingPP11[1].Tempo := S5T#1S700MS;
   TimeWeldingPP11[2].Tempo := S5T#1S;
   TimeWeldingPP11[3].Tempo := S5T#1S;
   TimeWeldingPP11[4].Tempo := S5T#1S;
   TimeWeldingPP11[5].Tempo := S5T#1S;
   TimeWeldingPP11[6].Tempo := S5T#1S;
   TimeWeldingPP11[7].Tempo := S5T#1S;
   TimeWeldingPP11[8].Tempo := S5T#1S;
   TimeWeldingPP11[9].Tempo := S5T#1S;
   TimeWeldingPP11[10].Tempo := S5T#1S;
   TimeWeldingPP11[11].Tempo := S5T#1S;
   TimeWeldingPP11[12].Tempo := S5T#1S;
   TimeWeldingPP11[13].Tempo := S5T#1S;
   TimeWeldingPP11[14].Tempo := S5T#1S;
   TimeWeldingPP11[15].Tempo := S5T#1S;
   TimeWeldingPP11[16].Tempo := S5T#1S;
   TimeWeldingPP11[17].Tempo := S5T#1S;
   TimeWeldingPP11[18].Tempo := S5T#1S;
   TimeWeldingPP11[19].Tempo := S5T#1S;
   TimeWeldingPP11[20].Tempo := S5T#1S;
   TimeWeldingPP12[1].Tempo := S5T#1S;
   TimeWeldingPP12[2].Tempo := S5T#1S;
   TimeWeldingPP12[3].Tempo := S5T#1S;
   TimeWeldingPP12[4].Tempo := S5T#1S;
   TimeWeldingPP12[5].Tempo := S5T#1S;
   TimeWeldingPP12[6].Tempo := S5T#1S;
   TimeWeldingPP12[7].Tempo := S5T#1S;
   TimeWeldingPP12[8].Tempo := S5T#1S;
   TimeWeldingPP12[9].Tempo := S5T#1S;
   TimeWeldingPP12[10].Tempo := S5T#1S;
   TimeWeldingPP12[11].Tempo := S5T#1S;
   TimeWeldingPP12[12].Tempo := S5T#1S;
   TimeWeldingPP12[13].Tempo := S5T#1S;
   TimeWeldingPP12[14].Tempo := S5T#1S;
   TimeWeldingPP12[15].Tempo := S5T#1S;
   TimeWeldingPP12[16].Tempo := S5T#1S;
   TimeWeldingPP12[17].Tempo := S5T#1S;
   TimeWeldingPP12[18].Tempo := S5T#1S;
   TimeWeldingPP12[19].Tempo := S5T#1S;
   TimeWeldingPP12[20].Tempo := S5T#1S;
   TimeWeldingPP13[1].Tempo := S5T#1S;
   TimeWeldingPP13[2].Tempo := S5T#1S;
   TimeWeldingPP13[3].Tempo := S5T#1S;
   TimeWeldingPP13[4].Tempo := S5T#1S;
   TimeWeldingPP13[5].Tempo := S5T#1S;
   TimeWeldingPP13[6].Tempo := S5T#1S;
   TimeWeldingPP13[7].Tempo := S5T#1S;
   TimeWeldingPP13[8].Tempo := S5T#1S;
   TimeWeldingPP13[9].Tempo := S5T#1S;
   TimeWeldingPP13[10].Tempo := S5T#1S;
   TimeWeldingPP13[11].Tempo := S5T#1S;
   TimeWeldingPP13[12].Tempo := S5T#1S;
   TimeWeldingPP13[13].Tempo := S5T#1S;
   TimeWeldingPP13[14].Tempo := S5T#1S;
   TimeWeldingPP13[15].Tempo := S5T#1S;
   TimeWeldingPP13[16].Tempo := S5T#1S;
   TimeWeldingPP13[17].Tempo := S5T#1S;
   TimeWeldingPP13[18].Tempo := S5T#1S;
   TimeWeldingPP13[19].Tempo := S5T#1S;
   TimeWeldingPP13[20].Tempo := S5T#1S;
   TimeWeldingPP14[1].Tempo := S5T#1S;
   TimeWeldingPP14[2].Tempo := S5T#1S;
   TimeWeldingPP14[3].Tempo := S5T#1S;
   TimeWeldingPP14[4].Tempo := S5T#1S;
   TimeWeldingPP14[5].Tempo := S5T#1S;
   TimeWeldingPP14[6].Tempo := S5T#1S;
   TimeWeldingPP14[7].Tempo := S5T#1S;
   TimeWeldingPP14[8].Tempo := S5T#1S;
   TimeWeldingPP14[9].Tempo := S5T#1S;
   TimeWeldingPP14[10].Tempo := S5T#1S;
   TimeWeldingPP14[11].Tempo := S5T#1S;
   TimeWeldingPP14[12].Tempo := S5T#1S;
   TimeWeldingPP14[13].Tempo := S5T#1S;
   TimeWeldingPP14[14].Tempo := S5T#1S;
   TimeWeldingPP14[15].Tempo := S5T#1S;
   TimeWeldingPP14[16].Tempo := S5T#1S;
   TimeWeldingPP14[17].Tempo := S5T#1S;
   TimeWeldingPP14[18].Tempo := S5T#1S;
   TimeWeldingPP14[19].Tempo := S5T#1S;
   TimeWeldingPP14[20].Tempo := S5T#1S;
   TimeWeldingPP15[1].Tempo := S5T#1S;
   TimeWeldingPP15[2].Tempo := S5T#1S;
   TimeWeldingPP15[3].Tempo := S5T#1S;
   TimeWeldingPP15[4].Tempo := S5T#1S;
   TimeWeldingPP15[5].Tempo := S5T#1S;
   TimeWeldingPP15[6].Tempo := S5T#1S;
   TimeWeldingPP15[7].Tempo := S5T#1S;
   TimeWeldingPP15[8].Tempo := S5T#1S;
   TimeWeldingPP15[9].Tempo := S5T#1S;
   TimeWeldingPP15[10].Tempo := S5T#1S;
   TimeWeldingPP15[11].Tempo := S5T#1S;
   TimeWeldingPP15[12].Tempo := S5T#1S;
   TimeWeldingPP15[13].Tempo := S5T#1S;
   TimeWeldingPP15[14].Tempo := S5T#1S;
   TimeWeldingPP15[15].Tempo := S5T#1S;
   TimeWeldingPP15[16].Tempo := S5T#1S;
   TimeWeldingPP15[17].Tempo := S5T#1S;
   TimeWeldingPP15[18].Tempo := S5T#1S;
   TimeWeldingPP15[19].Tempo := S5T#1S;
   TimeWeldingPP15[20].Tempo := S5T#1S;
   TimeWeldingPP16[1].Tempo := S5T#1S;
   TimeWeldingPP16[2].Tempo := S5T#1S;
   TimeWeldingPP16[3].Tempo := S5T#1S;
   TimeWeldingPP16[4].Tempo := S5T#1S;
   TimeWeldingPP16[5].Tempo := S5T#1S;
   TimeWeldingPP16[6].Tempo := S5T#1S;
   TimeWeldingPP16[7].Tempo := S5T#1S;
   TimeWeldingPP16[8].Tempo := S5T#1S;
   TimeWeldingPP16[9].Tempo := S5T#1S;
   TimeWeldingPP16[10].Tempo := S5T#1S;
   TimeWeldingPP16[11].Tempo := S5T#1S;
   TimeWeldingPP16[12].Tempo := S5T#1S;
   TimeWeldingPP16[13].Tempo := S5T#1S;
   TimeWeldingPP16[14].Tempo := S5T#1S;
   TimeWeldingPP16[15].Tempo := S5T#1S;
   TimeWeldingPP16[16].Tempo := S5T#1S;
   TimeWeldingPP16[17].Tempo := S5T#1S;
   TimeWeldingPP16[18].Tempo := S5T#1S;
   TimeWeldingPP16[19].Tempo := S5T#1S;
   TimeWeldingPP16[20].Tempo := S5T#1S;
   TimeWeldingPP17[1].Tempo := S5T#1S;
   TimeWeldingPP17[2].Tempo := S5T#1S;
   TimeWeldingPP17[3].Tempo := S5T#1S;
   TimeWeldingPP17[4].Tempo := S5T#1S;
   TimeWeldingPP17[5].Tempo := S5T#1S;
   TimeWeldingPP17[6].Tempo := S5T#1S;
   TimeWeldingPP17[7].Tempo := S5T#1S;
   TimeWeldingPP17[8].Tempo := S5T#1S;
   TimeWeldingPP17[9].Tempo := S5T#1S;
   TimeWeldingPP17[10].Tempo := S5T#1S;
   TimeWeldingPP17[11].Tempo := S5T#1S;
   TimeWeldingPP17[12].Tempo := S5T#1S;
   TimeWeldingPP17[13].Tempo := S5T#1S;
   TimeWeldingPP17[14].Tempo := S5T#1S;
   TimeWeldingPP17[15].Tempo := S5T#1S;
   TimeWeldingPP17[16].Tempo := S5T#1S;
   TimeWeldingPP17[17].Tempo := S5T#1S;
   TimeWeldingPP17[18].Tempo := S5T#1S;
   TimeWeldingPP17[19].Tempo := S5T#1S;
   TimeWeldingPP17[20].Tempo := S5T#1S;
   TimeWeldingPP18[1].Tempo := S5T#1S;
   TimeWeldingPP18[2].Tempo := S5T#1S;
   TimeWeldingPP18[3].Tempo := S5T#1S;
   TimeWeldingPP18[4].Tempo := S5T#1S;
   TimeWeldingPP18[5].Tempo := S5T#1S;
   TimeWeldingPP18[6].Tempo := S5T#1S;
   TimeWeldingPP18[7].Tempo := S5T#1S;
   TimeWeldingPP18[8].Tempo := S5T#1S;
   TimeWeldingPP18[9].Tempo := S5T#1S;
   TimeWeldingPP18[10].Tempo := S5T#1S;
   TimeWeldingPP18[11].Tempo := S5T#1S;
   TimeWeldingPP18[12].Tempo := S5T#1S;
   TimeWeldingPP18[13].Tempo := S5T#1S;
   TimeWeldingPP18[14].Tempo := S5T#1S;
   TimeWeldingPP18[15].Tempo := S5T#1S;
   TimeWeldingPP18[16].Tempo := S5T#1S;
   TimeWeldingPP18[17].Tempo := S5T#1S;
   TimeWeldingPP18[18].Tempo := S5T#1S;
   TimeWeldingPP18[19].Tempo := S5T#1S;
   TimeWeldingPP18[20].Tempo := S5T#1S;
   TimeWeldingPP19[1].Tempo := S5T#1S;
   TimeWeldingPP19[2].Tempo := S5T#1S;
   TimeWeldingPP19[3].Tempo := S5T#1S;
   TimeWeldingPP19[4].Tempo := S5T#1S;
   TimeWeldingPP19[5].Tempo := S5T#1S;
   TimeWeldingPP19[6].Tempo := S5T#1S;
   TimeWeldingPP19[7].Tempo := S5T#1S;
   TimeWeldingPP19[8].Tempo := S5T#1S;
   TimeWeldingPP19[9].Tempo := S5T#1S;
   TimeWeldingPP19[10].Tempo := S5T#1S;
   TimeWeldingPP19[11].Tempo := S5T#1S;
   TimeWeldingPP19[12].Tempo := S5T#1S;
   TimeWeldingPP19[13].Tempo := S5T#1S;
   TimeWeldingPP19[14].Tempo := S5T#1S;
   TimeWeldingPP19[15].Tempo := S5T#1S;
   TimeWeldingPP19[16].Tempo := S5T#1S;
   TimeWeldingPP19[17].Tempo := S5T#1S;
   TimeWeldingPP19[18].Tempo := S5T#1S;
   TimeWeldingPP19[19].Tempo := S5T#1S;
   TimeWeldingPP19[20].Tempo := S5T#1S;
   TimeWeldingPP20[1].Tempo := S5T#1S;
   TimeWeldingPP20[2].Tempo := S5T#1S;
   TimeWeldingPP20[3].Tempo := S5T#1S;
   TimeWeldingPP20[4].Tempo := S5T#1S;
   TimeWeldingPP20[5].Tempo := S5T#1S;
   TimeWeldingPP20[6].Tempo := S5T#1S;
   TimeWeldingPP20[7].Tempo := S5T#1S;
   TimeWeldingPP20[8].Tempo := S5T#1S;
   TimeWeldingPP20[9].Tempo := S5T#1S;
   TimeWeldingPP20[10].Tempo := S5T#1S;
   TimeWeldingPP20[11].Tempo := S5T#1S;
   TimeWeldingPP20[12].Tempo := S5T#1S;
   TimeWeldingPP20[13].Tempo := S5T#1S;
   TimeWeldingPP20[14].Tempo := S5T#1S;
   TimeWeldingPP20[15].Tempo := S5T#1S;
   TimeWeldingPP20[16].Tempo := S5T#1S;
   TimeWeldingPP20[17].Tempo := S5T#1S;
   TimeWeldingPP20[18].Tempo := S5T#1S;
   TimeWeldingPP20[19].Tempo := S5T#1S;
   TimeWeldingPP20[20].Tempo := S5T#1S;
END_DATA_BLOCK

DATA_BLOCK "DB180"	// DB 180
VERSION : 0.1
"FB24 - Gestione Mov Assi"
BEGIN
END_DATA_BLOCK

DATA_BLOCK "DB181"	// DB 181
VERSION : 0.1
"FB24 - Gestione Mov Assi"
BEGIN
END_DATA_BLOCK

DATA_BLOCK "DBWork2"	// DB 200
VERSION : 0.1
  STRUCT
   OffsetX_2 : DINT ;
   OffsetY_2 : DINT ;
   Riserva : BOOL ;
   Riserva1 : BOOL ;
   Riserva2 : BOOL ;
   Riserva3 : BOOL ;
   Riserva4 : BOOL ;
   Riserva5 : BOOL ;
   Riserva6 : BOOL ;
   Riserva7 : BOOL ;
   RivervaByte : BYTE ;
   RivervaByte1 : BYTE ;
   RivervaByte2 : BYTE ;
   RivervaByte3 : BYTE ;
   RivervaByte4 : BYTE ;
   RivervaByte5 : BYTE ;
   RivervaByte6 : BYTE ;
   RivervaByte7 : BYTE ;
   RiservaWord : WORD ;
   RiservaWord1 : WORD ;
   RiservaWord2 : WORD ;
   RiservaWord3 : WORD ;
   RiservaWord4 : WORD ;
   RiservaWord5 : WORD ;
   RiservaWord6 : WORD ;
   RiservaWord7 : WORD ;
   RiservaDWord : DWORD ;
   RiservaDWord1 : DWORD ;
   RiservaDWord2 : DWORD ;
   RiservaDWord3 : DWORD ;
   RiservaDWord4 : DWORD ;
   RiservaDWord5 : DWORD ;
   RiservaDWord6 : DWORD ;
   RiservaDWord7 : DWORD ;
   RiservaReal : REAL ;
   RiservaReal1 : REAL ;
   RiservaReal2 : REAL ;
   RiservaReal3 : REAL ;
   RiservaReal4 : REAL ;
   RiservaReal5 : REAL ;
   RiservaReal6 : REAL ;
   RiservaReal7 : REAL ;
  END_STRUCT ;	
BEGIN
END_DATA_BLOCK

ORGANIZATION_BLOCK "MAIN PROGRAM"	// OB 1
TITLE = "Main Program Sweep (Cycle)"
VERSION : 0.1
VAR_TEMP
  OB1_EV_CLASS : BYTE ;	//Bits 0-3 = 1 (Coming event), Bits 4-7 = 1 (Event class 1)
  OB1_SCAN_1 : BYTE ;	//1 (Cold restart scan 1 of OB 1), 3 (Scan 2-n of OB 1)
  OB1_PRIORITY : BYTE ;	//Priority of OB Execution
  OB1_OB_NUMBR : BYTE ;	//1 (Organization block 1, OB1)
  OB1_RESERVED_1 : BYTE ;	//Reserved for system
  OB1_RESERVED_2 : BYTE ;	//Reserved for system
  OB1_PREV_CYCLE : INT ;	//Cycle time of previous OB1 scan (milliseconds)
  OB1_MIN_CYCLE : INT ;	//Minimum cycle time of OB1 (milliseconds)
  OB1_MAX_CYCLE : INT ;	//Maximum cycle time of OB1 (milliseconds)
  OB1_DATE_TIME : DATE_AND_TIME ;	//Date and time OB1 started
END_VAR
BEGIN
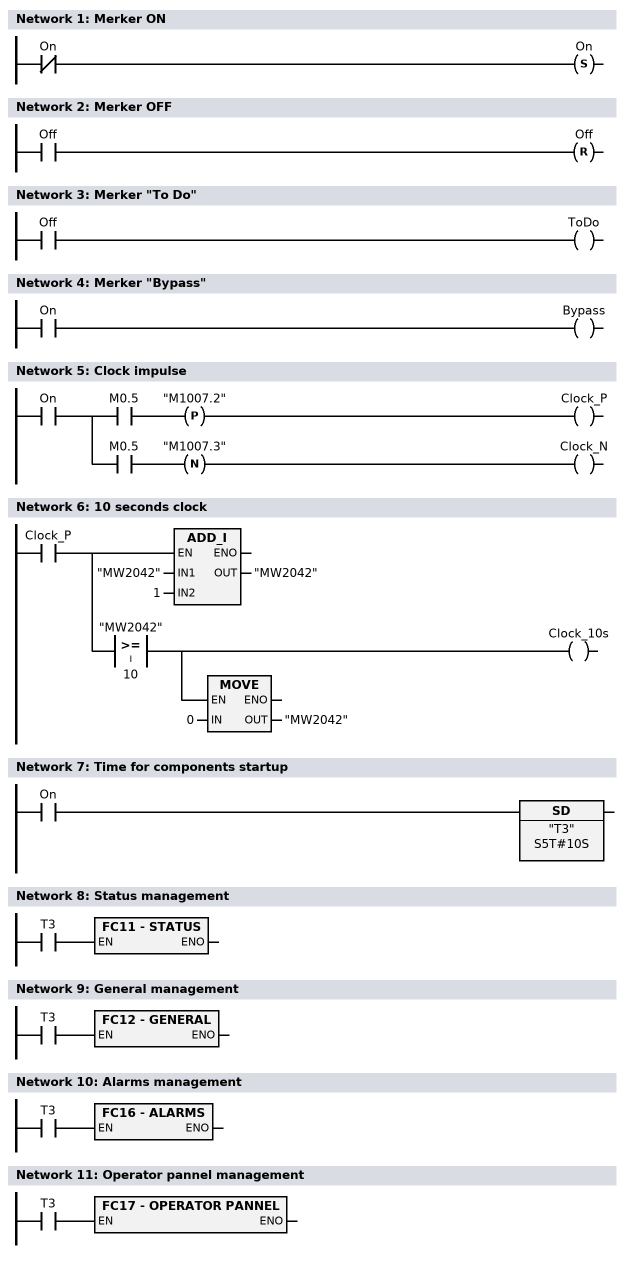
NETWORK
TITLE = Merker ON
      AN    "On";
      S     "On";
NETWORK
TITLE = Merker OFF
      A     "Off";
      R     "Off";
NETWORK
TITLE = Merker "To Do"
      A     "Off";
      =     "ToDo";
NETWORK
TITLE = Merker "Bypass"
      A     "On";
      =     "Bypass";
NETWORK
TITLE = Clock impulse
      A     "On";
      =     L 20.0;
      A     L 20.0;
      A     "M0.5";
      FP    "M1007.2";
      =     "Clock_P";
      A     L 20.0;
      A     "M0.5";
      FN    "M1007.3";
      =     "Clock_N";
NETWORK
TITLE = 10 seconds clock
      A     "Clock_P";
      =     L 20.0;
      A     L 20.0;
      JNB   _001;
      L     "MW2042";
      L     1;
      +I;
      T     "MW2042";
_001: NOP   0;
      A     L 20.0;
      A(;
      L     "MW2042";
      L     10;
      >=I;
      );
      =     L 20.1;
      A     L 20.1;
      BLD   102;
      =     "Clock_10s";
      A     L 20.1;
      JNB   _002;
      L     0;
      T     "MW2042";
_002: NOP   0;
NETWORK
TITLE = Time for components startup
      A     "On";
      L     S5T#10S;
      SD    "T3";
NETWORK
TITLE = Status management
      A     "T3";
      JNB   _003;
      CALL  "FC11 - STATUS";
_003: NOP   0;
NETWORK
TITLE = General management
      A     "T3";
      JNB   _004;
      CALL  "FC12 - GENERAL";
_004: NOP   0;
NETWORK
TITLE = Alarms management
      A     "T3";
      JNB   _005;
      CALL  "FC16 - ALARMS";
_005: NOP   0;
NETWORK
TITLE = Operator pannel management
      A     "T3";
      JNB   _006;
      CALL  "FC17 - OPERATOR PANNEL";
_006: NOP   0;
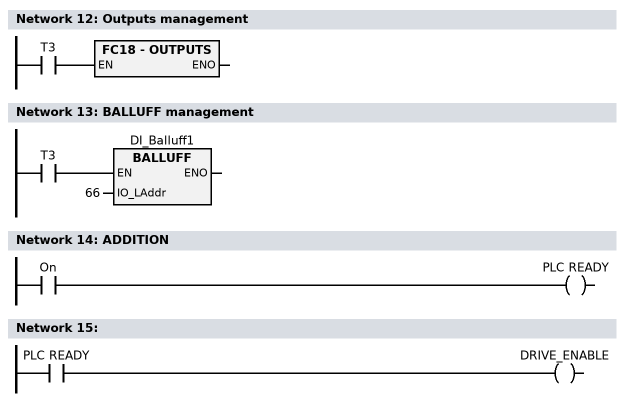
NETWORK
TITLE = Outputs management
      A     "T3";
      JNB   _007;
      CALL  "FC18 - OUTPUTS";
_007: NOP   0;
NETWORK
TITLE = BALLUFF management
      A     "T3";
      JNB   _008;
      CALL  "BALLUFF" , "DI_Balluff1" (
           IO_LAddr                 := 66);
_008: NOP   0;
NETWORK
TITLE = ADDITION
      A     "On";
      =     "PLC READY";
NETWORK
TITLE =
      A     "PLC READY";
      =     "DRIVE_ENABLE";
END_ORGANIZATION_BLOCK

ORGANIZATION_BLOCK "I/O_FLT1"	// OB 82
TITLE = "I/O Point Fault"
VERSION : 1.0
VAR_TEMP
  OB82_EV_CLASS : BYTE ;	// 16#39, Event class 3, entering event state, internal fault event
  OB82_FLT_ID : BYTE ;	// 16#XX, Fault identification code
  OB82_PRIORITY : BYTE ;	// 26/28 (Priority of 1 is lowest)
  OB82_OB_NUMBR : BYTE ;	// 82 (Organization block 82, OB82)
  OB82_RESERVED_1 : BYTE ;	// Reserved for system
  OB82_IO_FLAG : BYTE ;	// Input (01010100), Output (01010101)
  OB82_MDL_ADDR : INT ;	// Base address of module with fault
  OB82_MDL_DEFECT : BOOL ;	// Module defective
  OB82_INT_FAULT : BOOL ;	// Internal fault
  OB82_EXT_FAULT : BOOL ;	// External fault
  OB82_PNT_INFO : BOOL ;	// Point information
  OB82_EXT_VOLTAGE : BOOL ;	// External voltage low
  OB82_FLD_CONNCTR : BOOL ;	// Field wiring connector missing
  OB82_NO_CONFIG : BOOL ;	// Module has no configuration data
  OB82_CONFIG_ERR : BOOL ;	// Module has configuration error
  OB82_MDL_TYPE : BYTE ;	// Type of module
  OB82_SUB_NDL_ERR : BOOL ;	// Sub-Module is missing or has error
  OB82_COMM_FAULT : BOOL ;	// Communication fault
  OB82_MDL_STOP : BOOL ;	// Module is stopped
  OB82_WTCH_DOG_FLT : BOOL ;	// Watch dog timer stopped module
  OB82_INT_PS_FLT : BOOL ;	// Internal power supply fault
  OB82_PRIM_BATT_FLT : BOOL ;	// Primary battery is faulty
  OB82_BCKUP_BATT_FLT : BOOL ;	// Backup battery is faulty
  OB82_RESERVED_2 : BOOL ;	// Reserved for system
  OB82_RACK_FLT : BOOL ;	// Rack fault, only for bus interface module
  OB82_PROC_FLT : BOOL ;	// Processor fault
  OB82_EPROM_FLT : BOOL ;	// EPROM fault
  OB82_RAM_FLT : BOOL ;	// RAM fault
  OB82_ADU_FLT : BOOL ;	// ADC fault
  OB82_FUSE_FLT : BOOL ;	// Fuse fault
  OB82_HW_INTR_FLT : BOOL ;	// Hardware interrupt input faulty
  OB82_RESERVED_3 : BOOL ;	// Reserved for system
  OB82_DATE_TIME : DATE_AND_TIME ;	// Date and time OB82 started
END_VAR
BEGIN
NETWORK
TITLE =
END_ORGANIZATION_BLOCK

ORGANIZATION_BLOCK "RACK_FLT"	// OB 86
TITLE = "Loss Of Rack Fault"
VERSION : 0.1
VAR_TEMP
  OB86_EV_CLASS : BYTE ;	//16#38/39 Event class 3
  OB86_FLT_ID : BYTE ;	//16#C1/C4/C5, Fault identifcation code
  OB86_PRIORITY : BYTE ;	//Priority of OB Execution
  OB86_OB_NUMBR : BYTE ;	//86 (Organization block 86, OB86)
  OB86_RESERVED_1 : BYTE ;	//Reserved for system
  OB86_RESERVED_2 : BYTE ;	//Reserved for system
  OB86_MDL_ADDR : WORD ;	//Base address of IM module in rack with fault
  OB86_RACKS_FLTD : ARRAY  [0 .. 31 ] OF BOOL ;	//Racks in fault
  OB86_DATE_TIME : DATE_AND_TIME ;	//Date and time OB86 started
END_VAR
BEGIN
NETWORK
TITLE =
END_ORGANIZATION_BLOCK

ORGANIZATION_BLOCK "COMPLETE RESTART"	// OB 100
TITLE = "Complete Restart"
VERSION : 0.1
VAR_TEMP
  OB100_EV_CLASS : BYTE ;	//16#13, Event class 1, Entering event state, Event logged in diagnostic buffer
  OB100_STRTUP : BYTE ;	//16#81/82/83/84 Method of startup
  OB100_PRIORITY : BYTE ;	//Priority of OB Execution
  OB100_OB_NUMBR : BYTE ;	//100 (Organization block 100, OB100)
  OB100_RESERVED_1 : BYTE ;	//Reserved for system
  OB100_RESERVED_2 : BYTE ;	//Reserved for system
  OB100_STOP : WORD ;	//Event that caused CPU to stop (16#4xxx)
  OB100_STRT_INFO : DWORD ;	//Information on how system started
  OB100_DATE_TIME : DATE_AND_TIME ;	//Date and time OB100 started
END_VAR
BEGIN
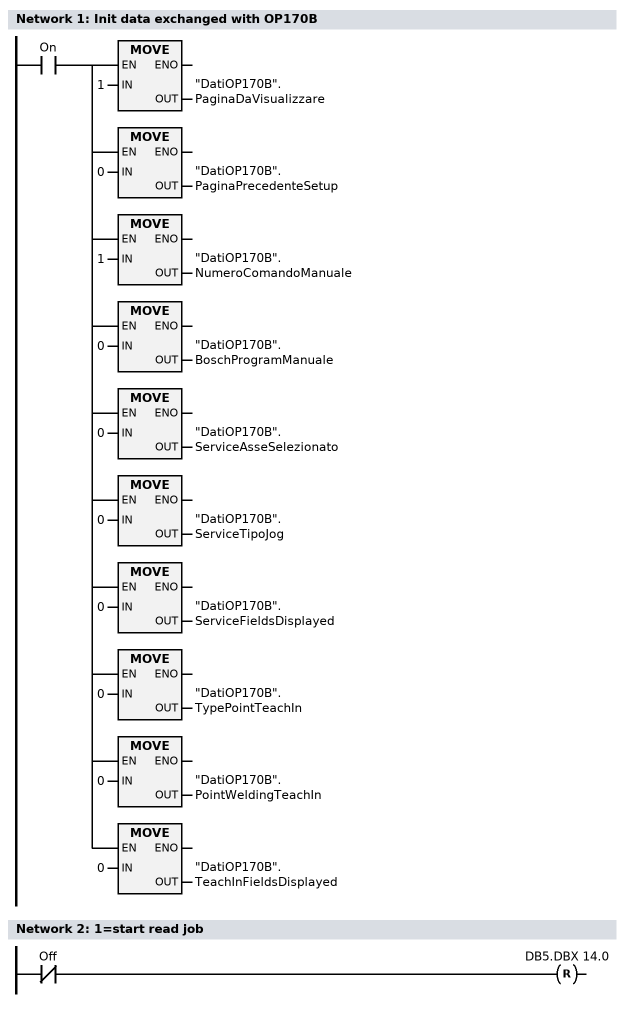
NETWORK
TITLE = Init data exchanged with OP170B
      A     "On";
      =     L 20.0;
      A     L 20.0;
      JNB   _001;
      L     1;
      T     "DatiOP170B".PaginaDaVisualizzare;
_001: NOP   0;
      A     L 20.0;
      JNB   _002;
      L     0;
      T     "DatiOP170B".PaginaPrecedenteSetup;
_002: NOP   0;
      A     L 20.0;
      JNB   _003;
      L     1;
      T     "DatiOP170B".NumeroComandoManuale;
_003: NOP   0;
      A     L 20.0;
      JNB   _004;
      L     0;
      T     "DatiOP170B".BoschProgramManuale;
_004: NOP   0;
      A     L 20.0;
      JNB   _005;
      L     0;
      T     "DatiOP170B".ServiceAsseSelezionato;
_005: NOP   0;
      A     L 20.0;
      JNB   _006;
      L     0;
      T     "DatiOP170B".ServiceTipoJog;
_006: NOP   0;
      A     L 20.0;
      JNB   _007;
      L     0;
      T     "DatiOP170B".ServiceFieldsDisplayed;
_007: NOP   0;
      A     L 20.0;
      JNB   _008;
      L     0;
      T     "DatiOP170B".TypePointTeachIn;
_008: NOP   0;
      A     L 20.0;
      JNB   _009;
      L     0;
      T     "DatiOP170B".PointWeldingTeachIn;
_009: NOP   0;
      A     L 20.0;
      JNB   _00a;
      L     0;
      T     "DatiOP170B".TeachInFieldsDisplayed;
_00a: NOP   0;
NETWORK
TITLE = 1=start read job
      AN    "Off";
      R     DB5.DBX 14.0;
END_ORGANIZATION_BLOCK

ORGANIZATION_BLOCK "MOD_ERR"	// OB 122
TITLE = "Module Access Error"
VERSION : 0.1
VAR_TEMP
  OB122_EV_CLASS : BYTE ;	//16#29, Event class 2, Entering event state, Internal fault event
  OB122_SW_FLT : BYTE ;	//16#XX Software error code
  OB122_PRIORITY : BYTE ;	//Priority of OB Execution
  OB122_OB_NUMBR : BYTE ;	//122 (Organization block 122, OB122)
  OB122_BLK_TYPE : BYTE ;	//16#88/8C/8E Type of block fault occured in
  OB122_MEM_AREA : BYTE ;	//Memory area where access error occured
  OB122_MEM_ADDR : WORD ;	//Memory address where access error occured
  OB122_BLK_NUM : WORD ;	//Block number in which error occured
  OB122_PRG_ADDR : WORD ;	//Program address where error occured
  OB122_DATE_TIME : DATE_AND_TIME ;	//Date and time OB1 started
END_VAR
BEGIN
NETWORK
TITLE =
END_ORGANIZATION_BLOCK

SYMBOL_TABLE
"Z10"	C 10	COUNTER	// Counter
"Z11"	C 11	COUNTER	// Counter
"Z12"	C 12	COUNTER	// Counter
"Z13"	C 13	COUNTER	// Counter
"DI_Balluff1"	DB 5	FB 20	// DB Instance of FB20
"DatiOP170B"	DB 7	DB 7	// PLC<->OP170B interface
"Timer"	DB 20	DB 20
"DBWork"	DB 21	DB 21
"coordinate"	DB 22	DB 22
"DB180"	DB 180	FB 24	// DB instance FB24 AsseY
"DB181"	DB 181	FB 24	// DB instance FB24 AsseX
"Asse_611U"	FB 16	FB 16	// Axis 611U management
"BALLUFF"	FB 20	FB 20	// BALLUFF Reader/Writer management
"FB24 - Gestione Mov Assi"	FB 24	FB 24	// GESTIONE ASSI STAZIONE
"NormalizzazioneAnalogico"	FC 7	FC 7	// Normalization of a analog value
"FC11 - STATUS"	FC 11	FC 11	// Sensors and proximity state
"FC12 - GENERAL"	FC 12	FC 12	// General management
"FC13 - MANUAL"	FC 13	FC 13	// Manual commands
"FC14 - AUTOMATIC"	FC 14	FC 14	// Automatic cycle management
"FC16 - ALARMS"	FC 16	FC 16	// Alarms management
"FC17 - OPERATOR PANNEL"	FC 17	FC 17	// Operator pannel management
"FC18 - OUTPUTS"	FC 18	FC 18	// Outputs management
"FC19 - REPOSITIONING"	FC 19	FC 19	// Repositioning management
"FC - AUTOMATIC"	FC 24	FC 24
"FC50 - TEACH-IN"	FC 50	FC 50
"FC51 - TYPE TOOL"	FC 51	FC 51
"FC52 - SYSTEM VISION"	FC 52	FC 52
"FC53 - REWORK"	FC 53	FC 53
"FC81 - GEST AXIS"	FC 81	FC 81	// Management axis
"FC117 - ERROR TOOL"	FC 117	FC 117
"TimeOut"	FC 800	FC 800	// Management TimeOut movimenti
"E0.0"	I 0.0	BOOL	// THERMAL SWTCH_ASPIRATOR_MTR
"E0.1"	I 0.1	BOOL	// 230 Vac power supply circuit braker
"E0.2"	I 0.2	BOOL	// 230 VAC PS CKT BRAKER
"E0.3"	I 0.3	BOOL	// Welding Machine OK
"E0.4"	I 0.4	BOOL	// Reserve
"E0.5"	I 0.5	BOOL	// AUXILIXARY ON
"DOOR CLOSE"	I 0.6	BOOL	// Reserve
"E0.7"	I 0.7	BOOL	// SAFETY BARRIER
"E1.0"	I 1.0	BOOL	// CYCLE_START
"E1.1"	I 1.1	BOOL	// AUTO_MANUAL
"E1.2"	I 1.2	BOOL	// COMPRESSED AIR
"E1.3"	I 1.3	BOOL	// AXIS RESET_POS
"E1.4"	I 1.4	BOOL	// Rotary table motor thermal switch
"E1.5"	I 1.5	BOOL	// LCK_UNLCK_DOORS_PB
"E1.6"	I 1.6	BOOL	// Reserve
"E1.7"	I 1.7	BOOL	// DRIVE TEMP
"E2.0"	I 2.0	BOOL	// STOP_CYCLE_PB
"E2.1"	I 2.1	BOOL	// Doors Closed & Locked
"E2.2"	I 2.2	BOOL	// Safety Barrier OK
"E2.3"	I 2.3	BOOL	// WELDING_TORCH_DWN
"E2.4"	I 2.4	BOOL	// WELDING_TORCH_UP
"E2.5"	I 2.5	BOOL	// ROTARY_TABLE_ZERO
"E2.6"	I 2.6	BOOL	// ROTARY_TABLE_ZERO1
"E2.7"	I 2.7	BOOL	// Reserve
"E3.0"	I 3.0	BOOL	// VEN DETECTOR_FWD
"E3.1"	I 3.1	BOOL	// VEN DETECTOR_REV
"E3.2"	I 3.2	BOOL	// VEN DETECTOR_DWN
"E3.3"	I 3.3	BOOL	// VEN DETECTOR_UP
"E3.4"	I 3.4	BOOL	// ROTARY_TABLE_CAM
"E3.5"	I 3.5	BOOL	// Reserve
"E3.6"	I 3.6	BOOL	// Reserve
"E3.7"	I 3.7	BOOL	// Reserve
"e5.0"	I 5.0	BOOL	// Lever Detector System - bit 0
"e5.1"	I 5.1	BOOL	// Lever Detector System - bit 1
"e5.2"	I 5.2	BOOL	// Lever Detector System - bit 2
"e5.3"	I 5.3	BOOL	// Lever Detector System - bit 3
"e5.4"	I 5.4	BOOL	// Lever Detector System - bit 4
"e5.5"	I 5.5	BOOL	// Lever Detector System - bit 5
"e5.6"	I 5.6	BOOL	// Lever Detector System - bit 6
"e5.7"	I 5.7	BOOL	// Lever Detector System - bit 7
"e6.0"	I 6.0	BOOL	// Lever Detector System - bit 8
"e6.1"	I 6.1	BOOL	// Lever Detector System - bit 9
"e6.2"	I 6.2	BOOL	// Lever Detector System - bit 10
"e6.3"	I 6.3	BOOL	// Lever Detector System - bit 11 - 12è13
"e6.4"	I 6.4	BOOL	// Lever Detector System - bit 12
"e6.5"	I 6.5	BOOL	// Lever Detector System - bit 13
"e6.6"	I 6.6	BOOL	// Lever Detector System - bit 14
"e6.7"	I 6.7	BOOL	// Lever Detector System - Vane Assy Total Number
"EXSTRACTOR_HIGH"	I 7.2	BOOL
"EXSTRACTOR_LOW"	I 7.3	BOOL
"TABLE_LCK_CYCLINDER_UP"	I 7.4	BOOL
"TABLE_LCK_CYCLINDER_DWN"	I 7.5	BOOL
"E32.0"	I 32.0	BOOL	// Push-button start cycle (on load position)
"E32.1"	I 32.1	BOOL	// Push button stop cycle
"E32.2"	I 32.2	BOOL	// Aut/Man Selector
"E32.3"	I 32.3	BOOL	// Reserve
"E32.4"	I 32.4	BOOL	// Reserve
"E32.5"	I 32.5	BOOL	// Lock/Unlock doors Push Button
"E32.6"	I 32.6	BOOL	// Reserve
"E32.7"	I 32.7	BOOL	// Air Presence
"E34.0"	I 34.0	BOOL	// Cam Table
"E34.1"	I 34.1	BOOL	// Reserve
"E34.2"	I 34.2	BOOL	// Reserve
"E34.3"	I 34.3	BOOL	// Reserve
"E34.4"	I 34.4	BOOL	// Table locker cylinder  up
"E34.5"	I 34.5	BOOL	// Table locker cylinder down
"E34.6"	I 34.6	BOOL	// Exstractor High
"E34.7"	I 34.7	BOOL	// Extractor Low
"E35.0"	I 35.0	BOOL	// Torch Welding low
"E35.1"	I 35.1	BOOL	// Torch Welding high
"E35.2"	I 35.2	BOOL	// Home Assy
"E35.3"	I 35.3	BOOL	// 1 --> PP1 on welding ; 0 --> PP2 on welding
"E35.4"	I 35.4	BOOL	// Detect components Control group High
"E35.5"	I 35.5	BOOL	// Detect components Control group Low
"E35.6"	I 35.6	BOOL	// Detect components Control group forward
"E35.7"	I 35.7	BOOL	// Detect components Control group backward
"E36.0"	I 36.0	BOOL	// Reserve not mounted
"E36.1"	I 36.1	BOOL	// Reserve not mounted
"E36.2"	I 36.2	BOOL	// Reserve not mounted
"E36.3"	I 36.3	BOOL	// Reserve not mounted
"E36.4"	I 36.4	BOOL	// Reserve not mounted
"E36.5"	I 36.5	BOOL	// Reserve not mounted
"E36.6"	I 36.6	BOOL	// Reserve not mounted
"E36.7"	I 36.7	BOOL	// Reserve not mounted
"E52.0"	I 52.0	BOOL	// Lever Detector System - bit 0
"E52.1"	I 52.1	BOOL	// Lever Detector System - bit 1
"E52.2"	I 52.2	BOOL	// Lever Detector System - bit 2
"E52.3"	I 52.3	BOOL	// Lever Detector System - bit 3
"E52.4"	I 52.4	BOOL	// Lever Detector System - bit 4
"E52.5"	I 52.5	BOOL	// Lever Detector System - bit 5
"E52.6"	I 52.6	BOOL	// Lever Detector System - bit 6
"E52.7"	I 52.7	BOOL	// Lever Detector System - bit 7
"E53.0"	I 53.0	BOOL	// Lever Detector System - bit 8
"E53.1"	I 53.1	BOOL	// Lever Detector System - bit 9
"E53.2"	I 53.2	BOOL	// Lever Detector System - bit 10
"E53.3"	I 53.3	BOOL	// Lever Detector System - bit 11 - 12è13
"E53.4"	I 53.4	BOOL	// Lever Detector System - bit 12
"E53.5"	I 53.5	BOOL	// Lever Detector System - bit 13
"E53.6"	I 53.6	BOOL	// Lever Detector System - bit 14
"E53.7"	I 53.7	BOOL	// Lever Detector System - Vane Assy Total Number
"E64.0"	I 64.0	BOOL	// VOSION SYSTEM OK
"E64.1"	I 64.1	BOOL	// Busy
"E64.2"	I 64.2	BOOL	// Or
"E64.3"	I 64.3	BOOL	// Error
"E64.4"	I 64.4	BOOL	// Gate
"E64.5"	I 64.5	BOOL	// Strobe trigger 0 out
"E64.6"	I 64.6	BOOL	// Strobe trigger 1 out
"E64.7"	I 64.7	BOOL	// DO0
"E65.0"	I 65.0	BOOL	// DO1
"E65.1"	I 65.1	BOOL	// DO2
"E65.2"	I 65.2	BOOL	// DO3
"E65.3"	I 65.3	BOOL	// DO4
"E65.4"	I 65.4	BOOL	// DO5
"E65.5"	I 65.5	BOOL	// DO6
"E65.6"	I 65.6	BOOL	// DO7
"E65.7"	I 65.7	BOOL	// DO8
"M0.0"	M 0.0	BOOL	// Clock 0,1 s
"M0.1"	M 0.1	BOOL	// Clock 0,2 s
"M0.2"	M 0.2	BOOL	// Clock 0,4 s
"M0.3"	M 0.3	BOOL	// Clock 0,5 s
"M0.4"	M 0.4	BOOL	// Clock 0,8 s
"M0.5"	M 0.5	BOOL	// Clock 1 s
"M0.6"	M 0.6	BOOL	// Clock 1,6 s
"M0.7"	M 0.7	BOOL	// Clock 2 s
"Off"	M 1.0	BOOL	// Merker always OFF
"On"	M 1.1	BOOL	// Merker always ON
"ToDo"	M 1.2	BOOL
"Bypass"	M 1.3	BOOL	// Merker that indicates a bypass forced of the code
"BypassPC"	M 1.4	BOOL	// Merker for bypass control handshake with PC supervision
"Clock_P"	M 1.5	BOOL	// Positiv pulse of clock
"Clock_N"	M 1.6	BOOL	// Negativ pulse of code
"Clock_10s"	M 1.7	BOOL	// 10 seconds clock
"BPSupervisor"	M 3.0	BOOL	// By Pass del supervisore
"Auxiliary_ON"	M 10.0	BOOL	// Auxiliary ON
"COMPRESSED_AIR"	M 10.1	BOOL	// Compressed Air
"SHIELDS_OK"	M 10.2	BOOL	// Schermi Chiusi e bloccati
"MACHINE_ON"	M 10.3	BOOL	// Machine OK
"START_POS"	M 11.0	BOOL	// Machine in initial positon
"START_POS_MEM"	M 11.1	BOOL	// mem initial position
"M11.2"	M 11.2	BOOL	// Manual Mode Selected
"SEMI"	M 11.3	BOOL	// Selezione modo semi automatico
"AUT"	M 11.4	BOOL	// Automatic Mode Selected
"START"	M 12.0	BOOL	// Start machine
"START_PULSE"	M 12.1	BOOL	// Pulse of start push-button
"SINGLE_CYCLE"	M 12.2	BOOL	// 1=ciclo singolo 0=ciclo continuo
"ALARM"	M 12.3	BOOL	// Alarm
"END_CYCLE"	M 12.4	BOOL	// Automatic cycle finished
"CmdMan_Av"	M 12.5	BOOL	// Forward manual command
"CmdMan_Ind"	M 12.6	BOOL	// Backward manual command
"STOP_BUTTON"	M 12.7	BOOL	// STATUS - stop button
"M13.0"	M 13.0	BOOL	// STATUS - Lock/Unlock doors Push Button
"M14.0"	M 14.0	BOOL	// Mem Lever Detector System - bit 0
"M14.1"	M 14.1	BOOL	// Mem Lever Detector System - bit 1
"M14.2"	M 14.2	BOOL	// Mem Lever Detector System - bit 2
"M14.3"	M 14.3	BOOL	// Mem Lever Detector System - bit 3
"M14.4"	M 14.4	BOOL	// Mem Lever Detector System - bit 4
"M14.5"	M 14.5	BOOL	// Mem Lever Detector System - bit 5
"M14.6"	M 14.6	BOOL	// Mem Lever Detector System - bit 6
"M14.7"	M 14.7	BOOL	// Mem Lever Detector System - bit 7
"M15.0"	M 15.0	BOOL	// Mem Lever Detector System - bit 8
"M15.1"	M 15.1	BOOL	// Mem Lever Detector System - bit 9
"M15.2"	M 15.2	BOOL	// Mem Lever Detector System - bit 10
"M15.3"	M 15.3	BOOL	// Mem Lever Detector System - bit 11
"M15.4"	M 15.4	BOOL	// Mem Lever Detector System - bit 12
"M15.5"	M 15.5	BOOL	// Mem Lever Detector System - bit 13
"M15.6"	M 15.6	BOOL	// Mem Detector System - bit0 select PP - E53.6
"M15.7"	M 15.7	BOOL	// Mem Detector System - bit1 select PP - E53.7
"M16.0"	M 16.0	BOOL	// mem Reworked Parts
"M16.1"	M 16.1	BOOL	// Disable Extractor if Rework
"M16.2"	M 16.2	BOOL	// Part on table 1 welding
"M16.3"	M 16.3	BOOL	// Part on Table 2 Welding
"M16.4"	M 16.4	BOOL	// Table can ROTATE
"M16.5"	M 16.5	BOOL	// Extractor can MOVE
"M16.6"	M 16.6	BOOL	// OK Extract
"M16.7"	M 16.7	BOOL	// Manual PAge Active
"M17.2"	M 17.2	BOOL	// Rework
"M17.3"	M 17.3	BOOL	// Vane no welding
"M17.4"	M 17.4	BOOL	// PP2 - OUT
"M17.5"	M 17.5	BOOL	// PP1 - OUT
"M17.6"	M 17.6	BOOL	// AUX - F R E E
"M17.7"	M 17.7	BOOL	// AUX - F R E E
"M18.0"	M 18.0	BOOL	// AUX - F R E E
"M18.1"	M 18.1	BOOL	// AUX - F R E E
"M18.2"	M 18.2	BOOL	// AUX - F R E E
"M18.3"	M 18.3	BOOL	// AUX - F R E E
"M18.4"	M 18.4	BOOL	// AUX - F R E E
"M18.5"	M 18.5	BOOL	// AUX - F R E E
"M18.6"	M 18.6	BOOL	// AUX - F R E E
"M18.7"	M 18.7	BOOL	// AUX - F R E E
"M19.0"	M 19.0	BOOL	// AUX - F R E E
"M19.1"	M 19.1	BOOL	// AUX - F R E E
"M19.2"	M 19.2	BOOL	// AUX - F R E E
"M19.3"	M 19.3	BOOL	// AUX - F R E E
"M19.4"	M 19.4	BOOL	// AUX - F R E E
"M19.5"	M 19.5	BOOL	// AUX - F R E E
"M19.6"	M 19.6	BOOL	// AUX - F R E E
"M19.7"	M 19.7	BOOL	// AUX - F R E E
"M20.0"	M 20.0	BOOL	// AUX - F R E E
"M20.1"	M 20.1	BOOL	// AUX - F R E E
"M20.2"	M 20.2	BOOL	// Presence of tool to assembly nozzle
"M20.3"	M 20.3	BOOL	// AUX - F R E E
"M20.4"	M 20.4	BOOL	// Tension OK
"M20.5"	M 20.5	BOOL	// AUX - F R E E
"M20.6"	M 20.6	BOOL	// AUX - F R E E
"M20.7"	M 20.7	BOOL	// AUX-Man
"M21.0"	M 21.0	BOOL	// STATUS - Mem Component pinched on Workrest - FC1
"Mem E34.5"	M 21.1	BOOL	// Mem Component pinched on Workrest - FC2
"M21.2"	M 21.2	BOOL	// AUX - F R E E
"M21.3"	M 21.3	BOOL	// AUX - F R E E
"M21.4"	M 21.4	BOOL	// Aux Alarm
"Warning"	M 21.5	BOOL	// Warning
"ResetAlarm"	M 21.6	BOOL	// Reset alarm
"Repos"	M 21.7	BOOL	// Repositioning
"M22.0"	M 22.0	BOOL	// STATUS - Table locker up
"M22.1"	M 22.1	BOOL	// STATUS - Table locker Down
"CmdMan_Av_Pulse"	M 22.2	BOOL	// Pulse of forward manual command
"CmdMan_Ind_Pulse"	M 22.3	BOOL	// Pulse of backward manual command
"M22.4"	M 22.4	BOOL	// Forward command
"M22.5"	M 22.5	BOOL	// Backward command
"CmdMan_Esg"	M 22.6	BOOL	// Memory of manual command executed
"CicloInCorso"	M 22.7	BOOL	// Automatic cycle in course
"M23.0"	M 23.0	BOOL	// Mem Start
"StopAEndCycle"	M 23.1	BOOL
"ChangeFunc"	M 23.2	BOOL	// Pulse change operation mode
"PresencePz"	M 23.3	BOOL
"SafetyBarrier_KO"	M 23.5	BOOL	// STATUS - Security bar KO
"M24.0"	M 24.0	BOOL	// STATUS - Torch Welding low
"M24.1"	M 24.1	BOOL	// STATUS - Torch Welding high
"M24.2"	M 24.2	BOOL	// STATUS -
"M24.3"	M 24.3	BOOL	// STATUS -
"M24.4"	M 24.4	BOOL	// STATUS - Cam table
"M24.5"	M 24.5	BOOL	// 1 --> PP1 on welding ;0 --> PP2 on welding
"M25.0"	M 25.0	BOOL	// Position Rotation 0°
"M25.1"	M 25.1	BOOL	// Position Rotation 180°
"M25.2"	M 25.2	BOOL	// Pos 0° e camma OK
"M25.3"	M 25.3	BOOL	// Pos 180° e camma OK
"M25.7"	M 25.7	BOOL	// Pulse Cam
"M26.1"	M 26.1	BOOL	// Table is FREE
"M26.2"	M 26.2	BOOL	// STATUS - System Detector Up
"M26.3"	M 26.3	BOOL	// STATUS - System Detector Lower
"M26.4"	M 26.4	BOOL	// STATUS - Detector work position
"M26.5"	M 26.5	BOOL	// STATUS - Detector park position
"M26.6"	M 26.6	BOOL	// STATUS - Exstractor High
"M26.7"	M 26.7	BOOL	// STATUS - Extractor low
"M28.0"	M 28.0	BOOL	// STATUS - DO1SYSTEM VISION
"M28.1"	M 28.1	BOOL	// STATUS - DO2 SYSTEM VISION
"M28.2"	M 28.2	BOOL	// STATUS - DO3 SYSTEM VISION
"M28.3"	M 28.3	BOOL	// STATUS - DO4 SYSTEM VISION
"M29.0"	M 29.0	BOOL	// STATUS - Run System Vision
"M29.1"	M 29.1	BOOL	// STATUS - Busy System Vision
"M29.2"	M 29.2	BOOL	// STATUS - OR System Vision
"M29.3"	M 29.3	BOOL	// STATUS - Error System Vision
"M29.4"	M 29.4	BOOL	// STATUS - Gate System Vision
"M29.6"	M 29.6	BOOL	// STATUS - DO1 SYSTEM VISION
"M29.7"	M 29.7	BOOL	// STATUS - DO0 SYSTEM VISION
"M30.0"	M 30.0	BOOL	// MAN - Table Rotation Forward
"M30.1"	M 30.1	BOOL	// MAN - Table Rotation Backward
"M30.2"	M 30.2	BOOL	// MAN - Jog + AsseY
"M30.3"	M 30.3	BOOL	// MAN - Jog - AsseY
"M30.4"	M 30.4	BOOL	// MAN - Jog + AsseX
"M30.5"	M 30.5	BOOL	// MAN - Jog - AsseX
"M30.6"	M 30.6	BOOL	// MAN - Forward SD
"M30.7"	M 30.7	BOOL	// MAN - Backward SD
"M31.0"	M 31.0	BOOL	// MAN - High SD
"M31.1"	M 31.1	BOOL	// MAN - Low SD
"M31.2"	M 31.2	BOOL	// MAN - High TW
"M31.3"	M 31.3	BOOL	// MAN - Low TW
"M31.4"	M 31.4	BOOL	// MAN - Extractor High
"M31.5"	M 31.5	BOOL	// MAN - Extractor down
"M31.6"	M 31.6	BOOL	// MAN - ON\OFF TW
"M31.7"	M 31.7	BOOL	// MAN - START/STOP WM
"M32.0"	M 32.0	BOOL	// Man  -  Start Torch W"elding
"M32.1"	M 32.1	BOOL	// MAN - Test Arco Gas Ok
"M32.2"	M 32.2	BOOL	// MAN - Test Arco Gas
"M32.3"	M 32.3	BOOL	// MAN - Torch Welding Temp Ok
"M32.4"	M 32.4	BOOL	// MAN - low table locker cylinder
"M32.5"	M 32.5	BOOL	// MAN - up table locker cylinder
"M32.6"	M 32.6	BOOL	// MAN - Welding
"M32.7"	M 32.7	BOOL	// MAN - Free
"M33.0"	M 33.0	BOOL	// MAN - Free
"M33.1"	M 33.1	BOOL	// MAN - Free
"M33.2"	M 33.2	BOOL	// MAN - Free
"M33.3"	M 33.3	BOOL	// MAN - Free
"M33.4"	M 33.4	BOOL	// MAN - Free
"M33.5"	M 33.5	BOOL	// MAN - Free
"M33.6"	M 33.6	BOOL	// MAN - Free
"M33.7"	M 33.7	BOOL	// MAN - Free
"M34.0"	M 34.0	BOOL	// MAN - Memory for rotation table
"M34.1"	M 34.1	BOOL	// MAN - Memory back rotation table
"M34.2"	M 34.2	BOOL	// MAN - Free
"M34.3"	M 34.3	BOOL	// MAN - Free
"M34.4"	M 34.4	BOOL	// MAN - Free
"M34.5"	M 34.5	BOOL	// MAN - Free
"M34.6"	M 34.6	BOOL	// MAN - Free
"M34.7"	M 34.7	BOOL	// MAN - Free
"M40.0"	M 40.0	BOOL	// RIP - Start repositioning
"M40.1"	M 40.1	BOOL	// RIP - Start reposit CamTable
"M40.2"	M 40.2	BOOL	// RIP - Cam Table
"M40.3"	M 40.3	BOOL	// RIP - System Detector vertical
"M40.4"	M 40.4	BOOL	// RIP - System Detector horizontal
"M40.5"	M 40.5	BOOL	// RIP - torch welding
"M40.6"	M 40.6	BOOL	// RIP - estractor
"M40.7"	M 40.7	BOOL	// RIP - Axis X and Y
"M41.0"	M 41.0	BOOL	// RIP - low table locker cylinder
"M41.1"	M 41.1	BOOL	// RIP - up table locker cylinder
"M41.2"	M 41.2	BOOL	// RIP - Free
"M41.3"	M 41.3	BOOL	// RIP - Free
"M41.4"	M 41.4	BOOL	// RIP - Free
"M41.5"	M 41.5	BOOL	// RIP - Free
"M41.6"	M 41.6	BOOL	// RIP - Free
"M41.7"	M 41.7	BOOL	// RIP - Free
"M42.0"	M 42.0	BOOL	// RIP - Free
"M42.1"	M 42.1	BOOL	// RIP - Table locker
"M42.2"	M 42.2	BOOL	// RIP - Free
"M42.3"	M 42.3	BOOL	// RIP - Free
"M42.4"	M 42.4	BOOL	// RIP - Free
"M42.5"	M 42.5	BOOL	// RIP - Free
"M42.6"	M 42.6	BOOL	// RIP - Free
"M42.7"	M 42.7	BOOL	// RIP - Free
"M50.0"	M 50.0	BOOL	// AUT - Table forward Side A
"M50.1"	M 50.1	BOOL	// AUT - Table backward Side B
"M50.2"	M 50.2	BOOL	// AUT - System Detector Forward
"M50.3"	M 50.3	BOOL	// AUT - System Detector Backward
"M50.4"	M 50.4	BOOL	// AUT - System Detector Low
"M50.5"	M 50.5	BOOL	// AUT - System Detector High
"M50.6"	M 50.6	BOOL	// AUT - welding down
"M50.7"	M 50.7	BOOL	// AUT - welding up
"M51.0"	M 51.0	BOOL	// AUT - Free
"M51.1"	M 51.1	BOOL	// AUT - Free
"M51.2"	M 51.2	BOOL	// AUT - Free
"M51.3"	M 51.3	BOOL	// AUT - Estractor High
"M51.4"	M 51.4	BOOL	// AUT - Estractor Low
"M51.5"	M 51.5	BOOL	// AUT - Free
"M51.6"	M 51.6	BOOL	// AUT - Free
"M51.7"	M 51.7	BOOL	// AUT - Free
"M52.0"	M 52.0	BOOL	// AUT -Temp  welding OK
"M52.1"	M 52.1	BOOL	// AUT - welding now
"M52.2"	M 52.2	BOOL	// AUT - Trigger System Vision
"M52.3"	M 52.3	BOOL	// AUT - ligth up
"M52.4"	M 52.4	BOOL	// AUT - Test Arc
"M52.5"	M 52.5	BOOL	// AUT - Test Arc Gas Ok
"M52.6"	M 52.6	BOOL	// AUT - low table locker cylinder
"M52.7"	M 52.7	BOOL	// AUT - up table locker cylinder
"M53.0"	M 53.0	BOOL	// AUT - Table locker Up
"M53.1"	M 53.1	BOOL	// AUT - Table locker Down
"M60.0"	M 60.0	BOOL	// STEP - 1:Table Forward
"M60.1"	M 60.1	BOOL	// STEP - 2:System Detector Forward
"M60.2"	M 60.2	BOOL	// STEP 3- System Detector Low
"M60.3"	M 60.3	BOOL	// STEP - 3 Check Nozzle Component
"M60.4"	M 60.4	BOOL	// STEP - 5 System detector High
"M60.5"	M 60.5	BOOL	// STEP 6 - System Detector Bacward
"M60.6"	M 60.6	BOOL	// STEP -7 welding down on point
"M60.7"	M 60.7	BOOL	// STEP - welding OK
"M61.0"	M 61.0	BOOL	// STEP - All welding is effectuated
"M61.1"	M 61.1	BOOL	// STEP - Photo Executed
"M61.2"	M 61.2	BOOL	// STEP - Axis in position 0
"M61.3"	M 61.3	BOOL	// STEP - point for welding receive
"M61.4"	M 61.4	BOOL	// STEP - welding up after work
"M61.5"	M 61.5	BOOL	// STEP - Welding in progress
"M61.6"	M 61.6	BOOL	// STEP - Start Rotation Table
"M61.7"	M 61.7	BOOL	// STEP - Photo without error
"M62.0"	M 62.0	BOOL	// STEP - Mem Reset Table
"M62.1"	M 62.1	BOOL	// STEP - Free
"M62.2"	M 62.2	BOOL	// STEP - Table cylinder up
"M62.3"	M 62.3	BOOL	// STEP - Free
"M62.4"	M 62.4	BOOL	// STEP - Free
"M62.5"	M 62.5	BOOL	// STEP - Free
"M62.6"	M 62.6	BOOL	// STEP - Free
"M62.7"	M 62.7	BOOL	// STEP - Photo Executed
"M63.0"	M 63.0	BOOL	// STEP - Nozzle Extracted
"M63.1"	M 63.1	BOOL	// STEP - Table Cylinder Low
"M63.6"	M 63.6	BOOL	// STEP - receive point photo
"M66.0"	M 66.0	BOOL	// STEP - photo 1 is NO good
"M66.1"	M 66.1	BOOL	// STEP - photo 2 is NO good
"M66.4"	M 66.4	BOOL	// STEP - Axis in position
"M66.6"	M 66.6	BOOL	// STEP - Execute 2th photo
"M66.7"	M 66.7	BOOL	// STEP - All photo is NO Good
"M67.0"	M 67.0	BOOL	// STEP - Axis Y in position
"M67.1"	M 67.1	BOOL	// STEP - Axis X in position
"M70.0"	M 70.0	BOOL	// Nozzle components Ok
"M70.1"	M 70.1	BOOL	// memNozzle-components Ok
"M70.2"	M 70.2	BOOL	// Component of Nozzle KO
"M70.3"	M 70.3	BOOL	// error assembling su PP1
"M70.4"	M 70.4	BOOL	// error assembling su PP2
"M71.0"	M 71.0	BOOL	// System Detector in Pos initial
"M72.0"	M 72.0	BOOL	// ready for welding
"M73.0"	M 73.0	BOOL	// Enable velocity for repositioning
"M74.0"	M 74.0	BOOL	// Output SV enable
"M74.1"	M 74.1	BOOL	// piece good
"M74.2"	M 74.2	BOOL	// piece reject
"M75.0"	M 75.0	BOOL	// Enable movement axis for teach in
"M75.1"	M 75.1	BOOL	// TeachIn OK
"M76.0"	M 76.0	BOOL	// position welding receive
"MEM Welding Machine OK"	M 80.0	BOOL
"Type_PP1"	M 90.0	BOOL	// PP1-10 presence
"Type_PP2"	M 90.1	BOOL	// presence PP2 -11 welding
"Type_PP3"	M 90.2	BOOL	// presence PP3 - 9welding
"Type_PP4"	M 90.3	BOOL	// presence PP4 - 13 Welding
"AUT STEP 1"	M 160.0	BOOL
"AUT STEP 2"	M 160.1	BOOL
"AUT STEP 3"	M 160.2	BOOL
"AUT STEP 4"	M 160.3	BOOL
"AUT STEP 5"	M 160.4	BOOL
"AUT STEP 6"	M 160.5	BOOL
"AUT STEP 7"	M 160.6	BOOL
"AUT STEP 8"	M 160.7	BOOL
"AUT STEP 9"	M 161.0	BOOL
"AUT STEP10"	M 161.1	BOOL
"AUT STEP11"	M 161.2	BOOL
"AUT STEP12"	M 161.3	BOOL
"AUT STEP13"	M 161.4	BOOL
"AUT STEP14"	M 161.5	BOOL
"AUT STEP15"	M 161.6	BOOL
"AUT STEP16"	M 161.7	BOOL
"AUT STEP17"	M 162.0	BOOL
"AUT STEP18"	M 162.1	BOOL
"AUT STEP19"	M 162.2	BOOL
"AUT STEP20"	M 162.3	BOOL
"AUT STEP21"	M 162.4	BOOL
"AUT STEP22"	M 162.5	BOOL
"AUT STEP23"	M 162.6	BOOL
"AUT STEP24"	M 162.7	BOOL
"AUT STEP25"	M 163.0	BOOL
"AUT STEP26"	M 163.1	BOOL
"AUT STEP27"	M 163.2	BOOL
"AUT STEP28"	M 163.3	BOOL
"AUT STEP29"	M 163.4	BOOL
"AUT STEP30"	M 163.5	BOOL
"Clock 0.5 S"	M 200.3	BOOL
"Clock 1s"	M 200.5	BOOL
"M254.0"	M 254.0	BOOL	// Front Command HOME
"M254.1"	M 254.1	BOOL	// Front Command END
"M256.0"	M 256.0	BOOL	// Pulse
"M256.2"	M 256.2	BOOL	// Pulse
"M256.6"	M 256.6	BOOL	// Pulse
"M256.7"	M 256.7	BOOL	// Pulse
"M340.0"	M 340.0	BOOL	// AXIS Y:STOP MOVE
"M340.1"	M 340.1	BOOL	// AXIS Y:START POSITIONING
"M340.2"	M 340.2	BOOL	// AXIS Y:START SEARCH HOME
"M340.3"	M 340.3	BOOL	// AXIS Y:START POSITIONING ON HOME
"M340.4"	M 340.4	BOOL	// AXIS X:COMMAND JOG PLUS
"M340.5"	M 340.5	BOOL	// AXIS X:COMANDO JOG LESS
"M341.0"	M 341.0	BOOL	// AXIS Y:ACHIEVED LOCATION
"M341.1"	M 341.1	BOOL	// AXIS Y:REFERED AXIS
"M341.2"	M 341.2	BOOL	// AXIS Y:AXIS LOCATION ON HOME
"M341.3"	M 341.3	BOOL	// AXIS Y:AXIS STOP NONE COMMAND PROGRESS
"M341.4"	M 341.4	BOOL	// AXIS Y:SETTING SETTING IN MOTION OK
"M341.5"	M 341.5	BOOL	// AXIS Y:ALLRM SETTING IN MOTION
"M342.0"	M 342.0	BOOL	// AXIS Y:AXIS ON CAM OF  REFERENCE
"M342.1"	M 342.1	BOOL	// AXIS Y:AXIS ON OVER RACE NEGATIVE HARDWARE
"M342.2"	M 342.2	BOOL	// AXIS Y:AXIS ON OVER RACE POSITIVE HARDWARE
"M342.3"	M 342.3	BOOL	// AXIS Y:COMMAND BRAKE PARKING
"M342.4"	M 342.4	BOOL	// AXIS Y:AXIS ON OVER RACE NEGATIVE SOFTWARE
"M342.5"	M 342.5	BOOL	// AXIS Y:AXIS ON OVER RACE POSITIVE SOFTWARE
"M342.6"	M 342.6	BOOL	// AXIS Y:POSSIBLE MOVE AXIS
"M342.7"	M 342.7	BOOL	// AXIS Y:INITIAL LOCATION AXIS
"M343.0"	M 343.0	BOOL	// AXIS Y:START POSITIONING INCREMENTAL
"M346.0"	M 346.0	BOOL	// AXIS X:STOP MOVE
"M346.1"	M 346.1	BOOL	// AXIS X:START POSITIONING
"M346.2"	M 346.2	BOOL	// AXIS X:START SEARCH HOME
"M346.3"	M 346.3	BOOL	// AXIS X:START POSITIONING ON HOME
"M346.4"	M 346.4	BOOL	// AXIS Y:COMMAND JOG PLUS
"M346.5"	M 346.5	BOOL	// AXIS Y:COMANDO JOG LESS
"M347.0"	M 347.0	BOOL	// AXIS X:ACHIEVED LOCATION
"M347.1"	M 347.1	BOOL	// AXIS X:REFERED AXIS
"M347.2"	M 347.2	BOOL	// AXIS X:AXIS LOCATION ON HOME
"M347.3"	M 347.3	BOOL	// AXIS X:AXIS STOP NONE COMMAND PROGRESS
"M347.4"	M 347.4	BOOL	// AXIS X:SETTING SETTING IN MOTION OK
"M347.5"	M 347.5	BOOL	// AXIS X:ALLRM SETTING IN MOTION
"M348.0"	M 348.0	BOOL	// AXIS X:AXIS ON CAM OF  REFERENCE
"M348.1"	M 348.1	BOOL	// AXIS X:AXIS ON OVER RACE NEGATIVE HARDWARE
"M348.2"	M 348.2	BOOL	// AXIS X:AXIS ON OVER RACE POSITIVE HARDWARE
"M348.3"	M 348.3	BOOL	// AXIS X:COMMAND BRAKE PARKING
"M348.4"	M 348.4	BOOL	// AXIS X:AXIS ON OVER RACE NEGATIVE SOFTWARE
"M348.5"	M 348.5	BOOL	// AXIS X:AXIS ON OVER RACE POSITIVE SOFTWARE
"M348.6"	M 348.6	BOOL	// AXIS X:POSSIBLE MOVE AXIS
"M348.7"	M 348.7	BOOL	// AXIS X:INITIAL LOCATION AXIS
"M349.0"	M 349.0	BOOL	// AXIS X:START POSITIONING INCREMENTAL
"CkCameraPrimaSaldatura"	M 500.0	BOOL	// Abilita ciclo controllo camera prima di saldare
"CkCamOKPrimaSaldatura"	M 500.1	BOOL	// Controllo camera OK prima di saldare
"DisabCkCamPreSaldatura"	M 500.2	BOOL	// Disabilita controllo camera prima di saldare
"AppoFP_M500.3"	M 500.3	BOOL
"TriggerCam_PrimaDiSaldar"	M 500.4	BOOL
"M1000.0"	M 1000.0	BOOL	// AUX
"M1000.1"	M 1000.1	BOOL	// AUX
"M1000.2"	M 1000.2	BOOL	// AUX
"M1000.3"	M 1000.3	BOOL	// AUX
"M1000.4"	M 1000.4	BOOL	// AUX
"M1000.5"	M 1000.5	BOOL	// AUX
"M1000.6"	M 1000.6	BOOL	// AUX
"M1000.7"	M 1000.7	BOOL	// AUX
"M1001.0"	M 1001.0	BOOL	// AUX
"M1001.1"	M 1001.1	BOOL	// AUX
"M1001.2"	M 1001.2	BOOL	// AUX
"M1001.3"	M 1001.3	BOOL	// AUX
"M1001.4"	M 1001.4	BOOL	// AUX
"M1001.5"	M 1001.5	BOOL	// AUX
"M1001.6"	M 1001.6	BOOL	// AUX
"M1001.7"	M 1001.7	BOOL	// AUX
"M1002.0"	M 1002.0	BOOL	// AUX
"M1002.1"	M 1002.1	BOOL	// AUX
"M1002.2"	M 1002.2	BOOL	// AUX
"M1002.3"	M 1002.3	BOOL	// AUX
"M1002.4"	M 1002.4	BOOL	// AUX
"M1002.5"	M 1002.5	BOOL	// AUX
"M1002.6"	M 1002.6	BOOL	// AUX
"M1002.7"	M 1002.7	BOOL	// AUX
"M1003.0"	M 1003.0	BOOL	// AUX
"M1003.1"	M 1003.1	BOOL	// AUX
"M1003.2"	M 1003.2	BOOL	// AUX
"M1003.3"	M 1003.3	BOOL	// AUX
"M1003.4"	M 1003.4	BOOL	// AUX
"M1003.5"	M 1003.5	BOOL	// AUX
"M1003.6"	M 1003.6	BOOL	// AUX
"M1003.7"	M 1003.7	BOOL	// AUX
"M1004.0"	M 1004.0	BOOL	// AUX
"M1004.1"	M 1004.1	BOOL	// AUX
"M1004.2"	M 1004.2	BOOL	// AUX
"M1004.3"	M 1004.3	BOOL	// AUX
"M1004.4"	M 1004.4	BOOL	// AUX
"M1004.5"	M 1004.5	BOOL	// AUX
"M1004.6"	M 1004.6	BOOL	// AUX
"M1004.7"	M 1004.7	BOOL	// AUX
"M1005.0"	M 1005.0	BOOL	// AUX
"M1005.1"	M 1005.1	BOOL	// AUX
"M1005.2"	M 1005.2	BOOL	// AUX
"M1005.3"	M 1005.3	BOOL	// AUX
"M1005.4"	M 1005.4	BOOL	// AUX
"M1005.5"	M 1005.5	BOOL	// AUX
"M1005.6"	M 1005.6	BOOL	// AUX
"M1005.7"	M 1005.7	BOOL	// AUX
"M1006.0"	M 1006.0	BOOL	// AUX
"M1006.1"	M 1006.1	BOOL	// AUX
"M1006.2"	M 1006.2	BOOL	// AUX
"M1006.3"	M 1006.3	BOOL	// AUX
"M1006.4"	M 1006.4	BOOL	// AUX
"M1006.5"	M 1006.5	BOOL	// AUX
"M1006.6"	M 1006.6	BOOL	// AUX
"M1006.7"	M 1006.7	BOOL	// AUX
"M1007.0"	M 1007.0	BOOL	// AUX
"M1007.1"	M 1007.1	BOOL	// AUX
"M1007.2"	M 1007.2	BOOL	// AUX
"M1007.3"	M 1007.3	BOOL	// AUX
"M1007.4"	M 1007.4	BOOL	// AUX
"M1007.5"	M 1007.5	BOOL	// AUX
"M1007.6"	M 1007.6	BOOL	// AUX
"M1007.7"	M 1007.7	BOOL	// AUX
"M1008.0"	M 1008.0	BOOL	// AUX
"M1008.1"	M 1008.1	BOOL	// AUX
"M1008.2"	M 1008.2	BOOL	// AUX
"M1008.3"	M 1008.3	BOOL	// AUX
"M1008.4"	M 1008.4	BOOL	// AUX
"M1008.5"	M 1008.5	BOOL	// AUX
"M1008.6"	M 1008.6	BOOL	// AUX
"M1008.7"	M 1008.7	BOOL	// AUX
"M1009.0"	M 1009.0	BOOL	// AUX
"M1009.1"	M 1009.1	BOOL	// AUX
"M1009.2"	M 1009.2	BOOL	// AUX
"M1009.3"	M 1009.3	BOOL	// AUX
"M1009.4"	M 1009.4	BOOL	// AUX
"M1009.5"	M 1009.5	BOOL	// AUX
"M1009.6"	M 1009.6	BOOL	// AUX
"M1009.7"	M 1009.7	BOOL	// AUX
"FPAuxON_force_Axis_reset"	M 1900.0	BOOL
"Luce telecamera"	M 1900.2	BOOL
"AppoFP_M1900.3"	M 1900.3	BOOL
"Soffio Camera"	M 1900.4	BOOL
"Manual_cameralight_on"	M 1900.5	BOOL
"M2034.0"	M 2034.0	BOOL	// Key Start from pannell
"M2034.1"	M 2034.1	BOOL	// Key Finish from pannell
"M2034.2"	M 2034.2	BOOL	// Key Teach In from Pannell
"M2034.5"	M 2034.5	BOOL	// Key Enter teach from pannel
"M2034.6"	M 2034.6	BOOL	// Key Exit teach from pannel
"M2034.7"	M 2034.7	BOOL	// Key Rite from pannell
"M2035.0"	M 2035.0	BOOL	// Key Start from Teach In page
"M2035.1"	M 2035.1	BOOL	// Key Welding Run from pannel
"M2035.2"	M 2035.2	BOOL	// Key ACK on page 21 from pannell
"MB2046"	MB 2046	BYTE	// white byte
"MD30"	MD 30	DWORD	// DWORD Manual Commands
"MD100"	MD 100	DWORD	// temp
"MD588"	MD 588	DINT	// temporary for X point
"MD592"	MD 592	DINT	// temporary for X point
"MD596"	MD 596	DINT	// target X
"MD600"	MD 600	DINT	// target Y
"MD620"	MD 620	DWORD	// InsertPointX
"MD624"	MD 624	DWORD	// InsertPointY
"MD650"	MD 650	DINT	// axis X actual position
"MD654"	MD 654	DINT	// axis Y actual posiion
"SaldEffet"	MW 110	WORD	// number welding make
"MW120"	MW 120	INT	// number welding make
"MW300"	MW 300	INT	// number point to want go
"MW2042"	MW 2042	INT	// temp for clock
"MAIN PROGRAM"	OB 1	OB 1	// Main Program
"I/O_FLT1"	OB 82	OB 82	// I/O Point Fault 1
"RACK_FLT"	OB 86	OB 86	// Loss of Rack Fault
"COMPLETE RESTART"	OB 100	OB 100	// Complete Restart
"MOD_ERR"	OB 122	OB 122	// Module Access Error
"A0.0"	Q 0.0	BOOL	// Red Lamp
"A0.1"	Q 0.1	BOOL	// Yellow Lamp
"A0.2"	Q 0.2	BOOL	// Green Lamp
"A0.3"	Q 0.3	BOOL	// Lock doors relay
"A0.4"	Q 0.4	BOOL	// Simodrive Reset realy
"A0.5"	Q 0.5	BOOL	// Reserve
"A0.6"	Q 0.6	BOOL	// Reserve
"A0.7"	Q 0.7	BOOL	// Reserve
"A1.0"	Q 1.0	BOOL	// Enable Coral Vacuum
"A1.1"	Q 1.1	BOOL	// Test Gas Arco Pilota
"A1.2"	Q 1.2	BOOL	// Forward table rotation
"A1.3"	Q 1.3	BOOL	// Backward table rotation
"A1.4"	Q 1.4	BOOL	// Enable Axis X
"A1.5"	Q 1.5	BOOL	// Enable Axis Y
"A1.6"	Q 1.6	BOOL	// Start Welding
"A1.7"	Q 1.7	BOOL	// Ignition torch
"A2.0"	Q 2.0	BOOL	// Reserve
"A2.1"	Q 2.1	BOOL	// Reserve
"A2.2"	Q 2.2	BOOL	// Reserve
"A2.3"	Q 2.3	BOOL	// Reserve
"A2.4"	Q 2.4	BOOL	// Reserve
"A2.5"	Q 2.5	BOOL	// Reserve
"A2.6"	Q 2.6	BOOL	// Reserve
"A2.7"	Q 2.7	BOOL	// Reserve
"A3.0"	Q 3.0	BOOL	// Reserve
"A3.1"	Q 3.1	BOOL	// Reserve
"A3.2"	Q 3.2	BOOL	// Reserve
"A3.3"	Q 3.3	BOOL	// Reserve
"A3.4"	Q 3.4	BOOL	// Reserve
"A3.5"	Q 3.5	BOOL	// Reserve
"A3.6"	Q 3.6	BOOL	// Reserve
"A3.7"	Q 3.7	BOOL	// Reserve
"SIMODRIVE_RESET"	Q 12.0	BOOL
"BUZZER"	Q 12.1	BOOL
"Torch Welding Machin"	Q 12.2	BOOL	// Down
"Torch Welding MachinE"	Q 12.3	BOOL	// UP
"TABLE_LCKER_DWN"	Q 12.4	BOOL
"Table locker cylinder up"	Q 12.5	BOOL
"FWD_LEVER_DETECT_SYS"	Q 12.6	BOOL
"REV_LEVER_DETECT_SYS"	Q 12.7	BOOL
"UP_lever detector system"	Q 13.0	BOOL
"DW_lever detector sys"	Q 13.1	BOOL
"UP_Down _Extractor"	Q 13.2	BOOL
"_soffio_telecamera"	Q 13.3	BOOL
"DRIVE_ENABLE"	Q 13.5	BOOL
"ENABLE_Y_AXIS"	Q 13.6	BOOL
"ENABLE_X_AXIS"	Q 13.7	BOOL
"STOP_CYCLE_LAMP"	Q 14.3	BOOL
"START_CYCLE_LAMP"	Q 14.4	BOOL
"a14.5"	Q 14.5	BOOL
"ACCESES_BARRIER_LAMP"	Q 14.6	BOOL
"Enable Coral Vacuum"	Q 17.0	BOOL
"FWD_TABLE_ROTATION"	Q 17.1	BOOL
"REVERSE_TABLE_ROTATION"	Q 17.2	BOOL
"IGNITION_TORCH"	Q 17.5	BOOL
"START_WELDING"	Q 17.6	BOOL
"Test Gas Arc Pilota"	Q 17.7	BOOL
"PLC READY"	Q 18.0	BOOL	// ADDITION
"_Illumin_telecamera"	Q 18.1	BOOL
"PIECE_REFUSE"	Q 18.3	BOOL
"RED_LAMP"	Q 18.4	BOOL
"PIECE_GOOD"	Q 18.5	BOOL
"Lamp_Door_Locked"	Q 18.6	BOOL
"LOCK_DOORS_RELAY"	Q 18.7	BOOL
"A32.0"	Q 32.0	BOOL	// Lamp Start cycle
"A32.1"	Q 32.1	BOOL	// Lamp Stop cycle
"A32.2"	Q 32.2	BOOL	// Piece Good
"A32.3"	Q 32.3	BOOL	// Piece Refuse
"A32.4"	Q 32.4	BOOL	// Unlocked doors
"A32.5"	Q 32.5	BOOL	// Emergency Lamp
"A32.6"	Q 32.6	BOOL	// Access barrier Lamp
"A32.7"	Q 32.7	BOOL	// Buzzer
"A33.0"	Q 33.0	BOOL	// Reserve
"A33.1"	Q 33.1	BOOL	// Reserve
"A33.2"	Q 33.2	BOOL	// Reserve
"A33.3"	Q 33.3	BOOL	// Reserve
"A33.4"	Q 33.4	BOOL	// Reserve not mounted
"A33.5"	Q 33.5	BOOL	// Reserve not mounted
"A33.6"	Q 33.6	BOOL	// Reserve not mounted
"A33.7"	Q 33.7	BOOL	// Reserve not mounted
"A34.0"	Q 34.0	BOOL	// Forward lever detector System
"A34.1"	Q 34.1	BOOL	// Backward lever detector System
"A34.2"	Q 34.2	BOOL	// Down lever detector system
"A34.3"	Q 34.3	BOOL	// Up lever detector system
"A34.4"	Q 34.4	BOOL	// Down Torch Welding Machine
"A34.5"	Q 34.5	BOOL	// Up Torch Welding Machine
"A34.6"	Q 34.6	BOOL	// Down Extractor
"A34.7"	Q 34.7	BOOL	// Up Extractor
"A35.0"	Q 35.0	BOOL	// Table locker down
"A35.1"	Q 35.1	BOOL	// Table locker up
"A35.2"	Q 35.2	BOOL	// Reserve
"A35.3"	Q 35.3	BOOL	// Reserve
"A35.4"	Q 35.4	BOOL	// Reserve
"A35.5"	Q 35.5	BOOL	// Reserve
"A35.6"	Q 35.6	BOOL	// Reserve
"A35.7"	Q 35.7	BOOL	// Reserve
"A64.0"	Q 64.0	BOOL	// Reset
"A64.1"	Q 64.1	BOOL	// Trigger
"A64.2"	Q 64.2	BOOL	// Data Send Request
"A64.3"	Q 64.3	BOOL	// DI0
"A64.4"	Q 64.4	BOOL	// DI1
"A64.5"	Q 64.5	BOOL	// DI2
"A64.6"	Q 64.6	BOOL	// DI3
"A64.7"	Q 64.7	BOOL	// DI4
"A65.0"	Q 65.0	BOOL	// DI5
"A65.1"	Q 65.1	BOOL	// DI6
"A65.2"	Q 65.2	BOOL	// DI7
"A65.3"	Q 65.3	BOOL	// DI8
"A65.4"	Q 65.4	BOOL	// DI9
"A65.5"	Q 65.5	BOOL	// Reserve
"A65.6"	Q 65.6	BOOL	// Reserve
"A65.7"	Q 65.7	BOOL	// Reserve
"TON"	SFB 4	SFB 4	// Generate an On Delay
"READ_CLK"	SFC 1	SFC 1	// Read System Clock
"DPRD_DAT"	SFC 14	SFC 14	// Read Consistent Data of a Standard DP Slave
"DPWR_DAT"	SFC 15	SFC 15	// Write Consistent Data to a Standard DP Slave
"BLKMOV"	SFC 20	SFC 20	// Copy Variables
"FILL"	SFC 21	SFC 21	// Initialize a Memory Area
"CREAT_DB"	SFC 22	SFC 22	// Create Data Block
"DIS_AIRT"	SFC 41	SFC 41	// Delay the Higher Priority Interrupts and Asynchronous Errors
"EN_AIRT"	SFC 42	SFC 42	// Enable Higher Priority Interrupts and Asynchronous Errors
"STP"	SFC 46	SFC 46	// Change the CPU to STOP
"LGC_GADR"	SFC 49	SFC 49	// Query the Module Slot Belonging to a Logical Address
"RDSYSST"	SFC 51	SFC 51	// Read a System Status List or Partial List
"WR_REC"	SFC 58	SFC 58	// Write Data Record
"RD_REC"	SFC 59	SFC 59	// Read a Data Record
"T2"	T 2	TIMER
"T3"	T 3	TIMER	// Time for Component Start UP
"T10"	T 10	TIMER	// Delay
"T11"	T 11	TIMER
"T12"	T 12	TIMER	// delay next step
"T13"	T 13	TIMER	// Delay
"T14"	T 14	TIMER	// timer for delay KO
"T15"	T 15	TIMER	// Delay
"T16"	T 16	TIMER	// Delay
"T17"	T 17	TIMER	// timer delay
"T18"	T 18	TIMER	// Delay
"T19"	T 19	TIMER	// delay
"T20"	T 20	TIMER	// timer delay
"T21"	T 21	TIMER	// Time Test Arc
"T22"	T 22	TIMER	// Delay
"T23"	T 23	TIMER	// Timer for repositioning
"T24"	T 24	TIMER	// Delay make 2th photo
"T25"	T 25	TIMER	// delay
"T26"	T 26	TIMER	// time for reset output rotation table
"T27"	T 27	TIMER	// Timer for Executed Photo
"T28"	T 28	TIMER	// Delay for entry in teach in mode
"T29"	T 29	TIMER	// delay for reset both axis
"T30"	T 30	TIMER	// timer dealy
"T31"	T 31	TIMER	// MAN - time for welding
"T32"	T 32	TIMER	// MAN - time for welding UP
"T33"	T 33	TIMER	// Delay
"T34"	T 34	TIMER	// Time Test Arco
"T35"	T 35	TIMER	// Delay
"T36"	T 36	TIMER	// delay for cam not present
"T37"	T 37	TIMER	// Time Torch Welding Ok
"T38"	T 38	TIMER	// timer reset alarms axis X
"T39"	T 39	TIMER	// timer reset alarms axis Y
"T40"	T 40	TIMER	// Time Torch Welding Ok
"T41"	T 41	TIMER	// delay alarm air pressure
"T42"	T 42	TIMER	// Timer stop welding
"T43"	T 43	TIMER	// Timer welding Manual
"T44"	T 44	TIMER	// Delay
"T45"	T 45	TIMER	// timer for upgrade value
"T46"	T 46	TIMER	// delay enable axis Ytimer reset alarms axis X
"T47"	T 47	TIMER	// delay
"T48"	T 48	TIMER	// delay enable axis Ytimer reset alarms axis Y
"T50"	T 50	TIMER	// Delay
"T51"	T 51	TIMER
"T52"	T 52	TIMER	// wait after rotation table
"T53"	T 53	TIMER	// delay for chek camera point
"T54"	T 54	TIMER	// delay turn OFF Buzzer
"AssiOkXCamera"	T 55	TIMER	// controllo cam prima di saldare
"TempoEsecuzioneFoto"	T 56	TIMER
"T60"	T 60	TIMER	// Delay for entry in teach in mode
"T61"	T 61	TIMER	// delay go in position for 2th photo
"T62"	T 62	TIMER	// delay for axis in position
"T63"	T 63	TIMER	// Delay
"T90"	T 90	TIMER	// delay allarm for Simodrive
"VAT_1"	VAT 1	
"Coordinate_saldatura"	VAT 2	
"I/O System Vision"	VAT 3	
"Saldatrice"	VAT 4	
"VAT_12"	VAT 5	
"VAT_PUNTI_AVV"	VAT 6	
"VAT_PUNTI_AVV_2"	VAT 7	
"DB22_SaldaturaSilv"	VAT 8	
"DB22_Sald_PP1"	VAT 9	
"VAT_tool check"	VAT 10	
"VAT_Balluff"	VAT 11	
"ASSE_P"	VAT 12	
"DB22_Sald_PP3"	VAT 13	
"VAT_Point"	VAT 14	
"VAT_Point 16"	VAT 15	
"DB22_Sald_PP16"	VAT 16	
"VAT_17"	VAT 17	
"Tipo portapezzo"	VAT 18	
END_SYMBOL_TABLE

